KUKA KRL program: Milling_2_222.src

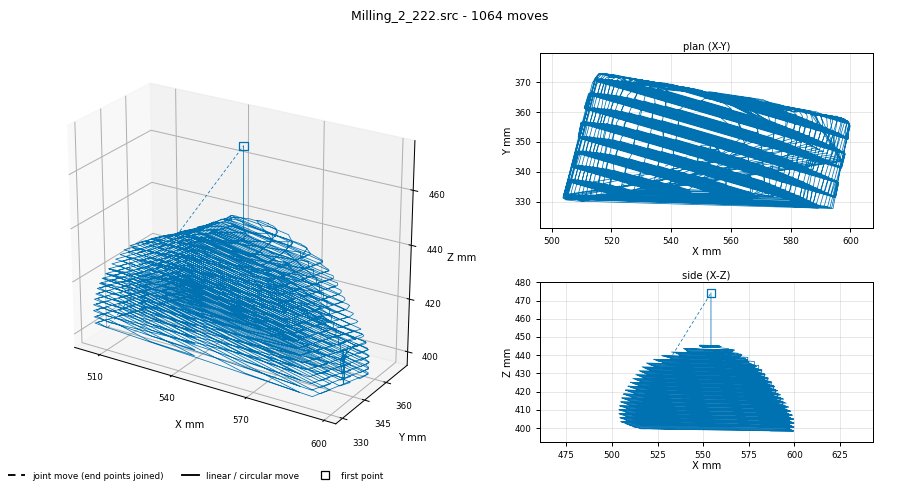
[picture p0: tool path of Milling_2_222.src, 1064 of 1066 moves have a stored position in this frame; points joined in program order, loops and branches not executed]
&ACCESS RVP
&REL 1
&PARAM TEMPLATE = C:\KRC\Roboter\Template\vorgabe
&PARAM EDITMASK = *
DEF Milling_2_222 ( )


;FOLD INI
;FOLD BASISTECH INI
GLOBAL INTERRUPT DECL 3 WHEN $STOPMESS==TRUE DO IR_STOPM ( )
INTERRUPT ON 3
BAS (#INITMOV,0 )
;ENDFOLD (BASISTECH INI)
;ENDFOLD (INI)

;FOLD STARTPOSITION - BASE IS 0, TOOL IS 5, SPEED IS 15%, POSITION IS A1 5,A2 -90,A3 100,A4 5,A5 -10,A6 -5,E1 0,E2 0,E3 0,E4 0
$BWDSTART = FALSE
PDAT_ACT = {VEL 15,ACC 100,APO_DIST 50}
FDAT_ACT = {TOOL_NO 5,BASE_NO 0,IPO_FRAME #BASE}
BAS (#PTP_PARAMS,15)
PTP  {A1 5,A2 -90,A3 100,A4 5,A5 -10,A6 -5,E1 0,E2 0,E3 0,E4 0}
;ENDFOLD

;FOLD LIN SPEED IS 0.1 m/sec, INTERPOLATION SETTINGS IN FOLD
$VEL.CP=0.1
$ADVANCE=3
;ENDFOLD

;FOLD COMMANDS IN FOLD. SELECT EDIT/FOLDS/OPEN ALL FOLDS TO DISPLAY
BAS(#VEL_PTP,2)
PTP {X 554.276, Y 348.908, Z 474.151, A -110.612, B 84.801, C -94.37, E1 0, E2 0, E3 0, E4 0, S 'B010'}
$VEL.CP=0.012
LIN {X 554.276, Y 348.908, Z 444.151, A -110.612, B 84.801, C -94.37, E1 0, E2 0, E3 0, E4 0}
LIN {X 558.607, Y 344.235, Z 444.41, A -110.612, B 84.801, C -94.37, E1 0, E2 0, E3 0, E4 0}
LIN {X 558.405, Y 342.44, Z 444.57, A -110.612, B 84.801, C -94.37, E1 0, E2 0, E3 0, E4 0}
LIN {X 559.721, Y 340.767, Z 444.67, A -110.612, B 84.801, C -94.37, E1 0, E2 0, E3 0, E4 0}
LIN {X 559.873, Y 339.853, Z 444.743, A -110.612, B 84.801, C -94.37, E1 0, E2 0, E3 0, E4 0}
LIN {X 557.875, Y 337.185, Z 445.034, A -110.612, B 84.801, C -94.37, E1 0, E2 0, E3 0, E4 0}
LIN {X 558.814, Y 334.358, Z 445.245, A -110.612, B 84.801, C -94.37, E1 0, E2 0, E3 0, E4 0}
LIN {X 549.81, Y 334.655, Z 445.508, A -110.612, B 84.801, C -94.37, E1 0, E2 0, E3 0, E4 0}
LIN {X 548.065, Y 334.808, Z 445.551, A -110.612, B 84.801, C -94.37, E1 0, E2 0, E3 0, E4 0}
LIN {X 547.985, Y 340.162, Z 445.098, A -110.612, B 84.801, C -94.37, E1 0, E2 0, E3 0, E4 0}
LIN {X 547.942, Y 340.376, Z 445.081, A -110.612, B 84.801, C -94.37, E1 0, E2 0, E3 0, E4 0}
LIN {X 549.959, Y 348.904, Z 444.29, A -110.612, B 84.801, C -94.37, E1 0, E2 0, E3 0, E4 0}
LIN {X 554.276, Y 348.908, Z 444.151, A -110.612, B 84.801, C -94.37, E1 0, E2 0, E3 0, E4 0}
LIN {X 556.311, Y 346.712, Z 444.273, A -110.612, B 84.801, C -94.37, E1 0, E2 0, E3 0, E4 0}
LIN {X 549.895, Y 348.583, Z 444.319, A -110.612, B 84.801, C -94.37, E1 0, E2 0, E3 0, E4 0}
LIN {X 548.877, Y 343.693, Z 444.768, A -110.612, B 84.801, C -94.37, E1 0, E2 0, E3 0, E4 0}
LIN {X 559.743, Y 340.524, Z 444.69, A -110.612, B 84.801, C -94.37, E1 0, E2 0, E3 0, E4 0}
LIN {X 558.354, Y 335.742, Z 445.142, A -110.612, B 84.801, C -94.37, E1 0, E2 0, E3 0, E4 0}
LIN {X 547.877, Y 338.798, Z 445.217, A -110.612, B 84.801, C -94.37, E1 0, E2 0, E3 0, E4 0}
LIN {X 563.989, Y 351.833, Z 443.591, A -110.612, B 84.801, C -94.37, E1 0, E2 0, E3 0, E4 0}
LIN {X 563.919, Y 351.649, Z 441.427, A -110.612, B 84.801, C -94.37, E1 0, E2 0, E3 0, E4 0}
LIN {X 565.535, Y 346.359, Z 441.825, A -110.612, B 84.801, C -94.37, E1 0, E2 0, E3 0, E4 0}
LIN {X 565.665, Y 346.192, Z 441.835, A -110.612, B 84.801, C -94.37, E1 0, E2 0, E3 0, E4 0}
LIN {X 567.236, Y 333.139, Z 442.897, A -110.612, B 84.801, C -94.37, E1 0, E2 0, E3 0, E4 0}
LIN {X 541.312, Y 334.209, Z 443.636, A -110.612, B 84.801, C -94.37, E1 0, E2 0, E3 0, E4 0}
LIN {X 539.137, Y 334.152, Z 443.71, A -110.612, B 84.801, C -94.37, E1 0, E2 0, E3 0, E4 0}
LIN {X 541.372, Y 343.839, Z 442.814, A -110.612, B 84.801, C -94.37, E1 0, E2 0, E3 0, E4 0}
LIN {X 540.702, Y 345.693, Z 442.677, A -110.612, B 84.801, C -94.37, E1 0, E2 0, E3 0, E4 0}
LIN {X 540.663, Y 347.231, Z 442.548, A -110.612, B 84.801, C -94.37, E1 0, E2 0, E3 0, E4 0}
LIN {X 540.807, Y 347.464, Z 442.523, A -110.612, B 84.801, C -94.37, E1 0, E2 0, E3 0, E4 0}
LIN {X 540.755, Y 349.434, Z 442.357, A -110.612, B 84.801, C -94.37, E1 0, E2 0, E3 0, E4 0}
LIN {X 541.559, Y 350.645, Z 442.228, A -110.612, B 84.801, C -94.37, E1 0, E2 0, E3 0, E4 0}
LIN {X 542.49, Y 357.115, Z 441.648, A -110.612, B 84.801, C -94.37, E1 0, E2 0, E3 0, E4 0}
LIN {X 543.459, Y 357.876, Z 441.552, A -110.612, B 84.801, C -94.37, E1 0, E2 0, E3 0, E4 0}
LIN {X 543.538, Y 358.445, Z 441.501, A -110.612, B 84.801, C -94.37, E1 0, E2 0, E3 0, E4 0}
LIN {X 541.559, Y 360.385, Z 441.399, A -110.612, B 84.801, C -94.37, E1 0, E2 0, E3 0, E4 0}
LIN {X 543.39, Y 361.216, Z 441.27, A -110.612, B 84.801, C -94.37, E1 0, E2 0, E3 0, E4 0}
LIN {X 544.179, Y 362.266, Z 441.155, A -110.612, B 84.801, C -94.37, E1 0, E2 0, E3 0, E4 0}
LIN {X 544.202, Y 362.541, Z 441.131, A -110.612, B 84.801, C -94.37, E1 0, E2 0, E3 0, E4 0}
LIN {X 544.848, Y 362.434, Z 441.119, A -110.612, B 84.801, C -94.37, E1 0, E2 0, E3 0, E4 0}
LIN {X 547.986, Y 363.741, Z 440.907, A -110.612, B 84.801, C -94.37, E1 0, E2 0, E3 0, E4 0}
LIN {X 548.585, Y 363.499, Z 440.909, A -110.612, B 84.801, C -94.37, E1 0, E2 0, E3 0, E4 0}
LIN {X 549.994, Y 363.669, Z 440.849, A -110.612, B 84.801, C -94.37, E1 0, E2 0, E3 0, E4 0}
LIN {X 551.281, Y 364.62, Z 440.727, A -110.612, B 84.801, C -94.37, E1 0, E2 0, E3 0, E4 0}
LIN {X 554.079, Y 364.139, Z 440.678, A -110.612, B 84.801, C -94.37, E1 0, E2 0, E3 0, E4 0}
LIN {X 554.813, Y 364.232, Z 440.647, A -110.612, B 84.801, C -94.37, E1 0, E2 0, E3 0, E4 0}
LIN {X 554.86, Y 363.85, Z 440.678, A -110.612, B 84.801, C -94.37, E1 0, E2 0, E3 0, E4 0}
LIN {X 557.614, Y 363.059, Z 440.657, A -110.612, B 84.801, C -94.37, E1 0, E2 0, E3 0, E4 0}
LIN {X 559.744, Y 361.401, Z 440.73, A -110.612, B 84.801, C -94.37, E1 0, E2 0, E3 0, E4 0}
LIN {X 560.566, Y 360.153, Z 440.81, A -110.612, B 84.801, C -94.37, E1 0, E2 0, E3 0, E4 0}
LIN {X 561.613, Y 359.2, Z 440.857, A -110.612, B 84.801, C -94.37, E1 0, E2 0, E3 0, E4 0}
LIN {X 563.919, Y 351.649, Z 441.427, A -110.612, B 84.801, C -94.37, E1 0, E2 0, E3 0, E4 0}
LIN {X 550.229, Y 363.842, Z 440.827, A -110.612, B 84.801, C -94.37, E1 0, E2 0, E3 0, E4 0}
LIN {X 560.058, Y 360.976, Z 440.756, A -110.612, B 84.801, C -94.37, E1 0, E2 0, E3 0, E4 0}
LIN {X 563.393, Y 354.816, Z 441.174, A -110.612, B 84.801, C -94.37, E1 0, E2 0, E3 0, E4 0}
LIN {X 542.631, Y 360.871, Z 441.323, A -110.612, B 84.801, C -94.37, E1 0, E2 0, E3 0, E4 0}
LIN {X 542.344, Y 355.768, Z 441.767, A -110.612, B 84.801, C -94.37, E1 0, E2 0, E3 0, E4 0}
LIN {X 565.078, Y 349.137, Z 441.603, A -110.612, B 84.801, C -94.37, E1 0, E2 0, E3 0, E4 0}
LIN {X 565.885, Y 343.715, Z 442.039, A -110.612, B 84.801, C -94.37, E1 0, E2 0, E3 0, E4 0}
LIN {X 541.583, Y 350.803, Z 442.214, A -110.612, B 84.801, C -94.37, E1 0, E2 0, E3 0, E4 0}
LIN {X 540.685, Y 345.878, Z 442.662, A -110.612, B 84.801, C -94.37, E1 0, E2 0, E3 0, E4 0}
LIN {X 566.796, Y 338.262, Z 442.474, A -110.612, B 84.801, C -94.37, E1 0, E2 0, E3 0, E4 0}
LIN {X 566.499, Y 333.162, Z 442.918, A -110.612, B 84.801, C -94.37, E1 0, E2 0, E3 0, E4 0}
LIN {X 540.83, Y 340.648, Z 443.103, A -110.612, B 84.801, C -94.37, E1 0, E2 0, E3 0, E4 0}
LIN {X 539.697, Y 335.792, Z 443.553, A -110.612, B 84.801, C -94.37, E1 0, E2 0, E3 0, E4 0}
LIN {X 545.888, Y 333.986, Z 443.508, A -110.612, B 84.801, C -94.37, E1 0, E2 0, E3 0, E4 0}
LIN {X 569.078, Y 353.533, Z 441.101, A -110.612, B 84.801, C -94.37, E1 0, E2 0, E3 0, E4 0}
LIN {X 569.009, Y 353.348, Z 438.936, A -110.612, B 84.801, C -94.37, E1 0, E2 0, E3 0, E4 0}
LIN {X 570.01, Y 350.644, Z 439.134, A -110.612, B 84.801, C -94.37, E1 0, E2 0, E3 0, E4 0}
LIN {X 571.217, Y 336.984, Z 440.258, A -110.612, B 84.801, C -94.37, E1 0, E2 0, E3 0, E4 0}
LIN {X 570.966, Y 336.181, Z 440.335, A -110.612, B 84.801, C -94.37, E1 0, E2 0, E3 0, E4 0}
LIN {X 570.983, Y 334.774, Z 440.454, A -110.612, B 84.801, C -94.37, E1 0, E2 0, E3 0, E4 0}
LIN {X 570.338, Y 332.582, Z 440.661, A -110.612, B 84.801, C -94.37, E1 0, E2 0, E3 0, E4 0}
LIN {X 534.018, Y 333.771, Z 441.723, A -110.612, B 84.801, C -94.37, E1 0, E2 0, E3 0, E4 0}
LIN {X 532.644, Y 333.742, Z 441.77, A -110.612, B 84.801, C -94.37, E1 0, E2 0, E3 0, E4 0}
LIN {X 535.31, Y 339.493, Z 441.195, A -110.612, B 84.801, C -94.37, E1 0, E2 0, E3 0, E4 0}
LIN {X 535.287, Y 341.092, Z 441.059, A -110.612, B 84.801, C -94.37, E1 0, E2 0, E3 0, E4 0}
LIN {X 537.309, Y 348.411, Z 440.371, A -110.612, B 84.801, C -94.37, E1 0, E2 0, E3 0, E4 0}
LIN {X 537.606, Y 348.945, Z 440.316, A -110.612, B 84.801, C -94.37, E1 0, E2 0, E3 0, E4 0}
LIN {X 537.307, Y 354.669, Z 439.838, A -110.612, B 84.801, C -94.37, E1 0, E2 0, E3 0, E4 0}
LIN {X 536.893, Y 356.232, Z 439.719, A -110.612, B 84.801, C -94.37, E1 0, E2 0, E3 0, E4 0}
LIN {X 536.949, Y 357.185, Z 439.636, A -110.612, B 84.801, C -94.37, E1 0, E2 0, E3 0, E4 0}
LIN {X 537.165, Y 357.599, Z 439.593, A -110.612, B 84.801, C -94.37, E1 0, E2 0, E3 0, E4 0}
LIN {X 538.343, Y 363.903, Z 439.019, A -110.612, B 84.801, C -94.37, E1 0, E2 0, E3 0, E4 0}
LIN {X 538.336, Y 363.912, Z 439.018, A -110.612, B 84.801, C -94.37, E1 0, E2 0, E3 0, E4 0}
LIN {X 537.831, Y 366.807, Z 438.788, A -110.612, B 84.801, C -94.37, E1 0, E2 0, E3 0, E4 0}
LIN {X 537.936, Y 366.972, Z 438.77, A -110.612, B 84.801, C -94.37, E1 0, E2 0, E3 0, E4 0}
LIN {X 539.378, Y 367.681, Z 438.664, A -110.612, B 84.801, C -94.37, E1 0, E2 0, E3 0, E4 0}
LIN {X 552.236, Y 366.051, Z 438.391, A -110.612, B 84.801, C -94.37, E1 0, E2 0, E3 0, E4 0}
LIN {X 554.008, Y 366.638, Z 438.284, A -110.612, B 84.801, C -94.37, E1 0, E2 0, E3 0, E4 0}
LIN {X 562.727, Y 364.468, Z 438.19, A -110.612, B 84.801, C -94.37, E1 0, E2 0, E3 0, E4 0}
LIN {X 566.199, Y 360.577, Z 438.41, A -110.612, B 84.801, C -94.37, E1 0, E2 0, E3 0, E4 0}
LIN {X 567.699, Y 358.885, Z 438.506, A -110.612, B 84.801, C -94.37, E1 0, E2 0, E3 0, E4 0}
LIN {X 569.005, Y 355.632, Z 438.741, A -110.612, B 84.801, C -94.37, E1 0, E2 0, E3 0, E4 0}
LIN {X 569.009, Y 353.348, Z 438.936, A -110.612, B 84.801, C -94.37, E1 0, E2 0, E3 0, E4 0}
LIN {X 567.859, Y 358.496, Z 438.534, A -110.612, B 84.801, C -94.37, E1 0, E2 0, E3 0, E4 0}
LIN {X 538.218, Y 367.141, Z 438.747, A -110.612, B 84.801, C -94.37, E1 0, E2 0, E3 0, E4 0}
LIN {X 538.244, Y 361.946, Z 439.189, A -110.612, B 84.801, C -94.37, E1 0, E2 0, E3 0, E4 0}
LIN {X 569.164, Y 352.928, Z 438.966, A -110.612, B 84.801, C -94.37, E1 0, E2 0, E3 0, E4 0}
LIN {X 570.368, Y 347.39, Z 439.4, A -110.612, B 84.801, C -94.37, E1 0, E2 0, E3 0, E4 0}
LIN {X 536.951, Y 357.136, Z 439.64, A -110.612, B 84.801, C -94.37, E1 0, E2 0, E3 0, E4 0}
LIN {X 537.304, Y 351.846, Z 440.079, A -110.612, B 84.801, C -94.37, E1 0, E2 0, E3 0, E4 0}
LIN {X 570.875, Y 342.055, Z 439.838, A -110.612, B 84.801, C -94.37, E1 0, E2 0, E3 0, E4 0}
LIN {X 571.155, Y 336.786, Z 440.277, A -110.612, B 84.801, C -94.37, E1 0, E2 0, E3 0, E4 0}
LIN {X 536.952, Y 346.762, Z 440.523, A -110.612, B 84.801, C -94.37, E1 0, E2 0, E3 0, E4 0}
LIN {X 535.523, Y 341.992, Z 440.975, A -110.612, B 84.801, C -94.37, E1 0, E2 0, E3 0, E4 0}
LIN {X 566.961, Y 332.823, Z 440.749, A -110.612, B 84.801, C -94.37, E1 0, E2 0, E3 0, E4 0}
LIN {X 546.398, Y 333.633, Z 441.339, A -110.612, B 84.801, C -94.37, E1 0, E2 0, E3 0, E4 0}
LIN {X 534.432, Y 337.123, Z 441.425, A -110.612, B 84.801, C -94.37, E1 0, E2 0, E3 0, E4 0}
LIN {X 574.468, Y 352.804, Z 438.807, A -110.612, B 84.801, C -94.37, E1 0, E2 0, E3 0, E4 0}
LIN {X 574.398, Y 352.62, Z 436.642, A -110.612, B 84.801, C -94.37, E1 0, E2 0, E3 0, E4 0}
LIN {X 574.985, Y 358.624, Z 436.112, A -110.612, B 84.801, C -94.37, E1 0, E2 0, E3 0, E4 0}
LIN {X 569.893, Y 363.529, Z 435.858, A -110.612, B 84.801, C -94.37, E1 0, E2 0, E3 0, E4 0}
LIN {X 568.224, Y 364.067, Z 435.865, A -110.612, B 84.801, C -94.37, E1 0, E2 0, E3 0, E4 0}
LIN {X 568.037, Y 364.329, Z 435.849, A -110.612, B 84.801, C -94.37, E1 0, E2 0, E3 0, E4 0}
LIN {X 567.581, Y 364.537, Z 435.846, A -110.612, B 84.801, C -94.37, E1 0, E2 0, E3 0, E4 0}
LIN {X 554.164, Y 366.346, Z 436.121, A -110.612, B 84.801, C -94.37, E1 0, E2 0, E3 0, E4 0}
LIN {X 553.733, Y 366.168, Z 436.15, A -110.612, B 84.801, C -94.37, E1 0, E2 0, E3 0, E4 0}
LIN {X 542.465, Y 368.047, Z 436.351, A -110.612, B 84.801, C -94.37, E1 0, E2 0, E3 0, E4 0}
LIN {X 540.849, Y 369.238, Z 436.301, A -110.612, B 84.801, C -94.37, E1 0, E2 0, E3 0, E4 0}
LIN {X 538.504, Y 369.469, Z 436.357, A -110.612, B 84.801, C -94.37, E1 0, E2 0, E3 0, E4 0}
LIN {X 537.187, Y 369.143, Z 436.427, A -110.612, B 84.801, C -94.37, E1 0, E2 0, E3 0, E4 0}
LIN {X 535.889, Y 368.249, Z 436.545, A -110.612, B 84.801, C -94.37, E1 0, E2 0, E3 0, E4 0}
LIN {X 534.308, Y 366.474, Z 436.746, A -110.612, B 84.801, C -94.37, E1 0, E2 0, E3 0, E4 0}
LIN {X 534.281, Y 366.405, Z 436.753, A -110.612, B 84.801, C -94.37, E1 0, E2 0, E3 0, E4 0}
LIN {X 534.584, Y 363.066, Z 437.028, A -110.612, B 84.801, C -94.37, E1 0, E2 0, E3 0, E4 0}
LIN {X 534.095, Y 360.828, Z 437.234, A -110.612, B 84.801, C -94.37, E1 0, E2 0, E3 0, E4 0}
LIN {X 533.835, Y 360.635, Z 437.259, A -110.612, B 84.801, C -94.37, E1 0, E2 0, E3 0, E4 0}
LIN {X 533.475, Y 357.247, Z 437.559, A -110.612, B 84.801, C -94.37, E1 0, E2 0, E3 0, E4 0}
LIN {X 533.725, Y 356.099, Z 437.649, A -110.612, B 84.801, C -94.37, E1 0, E2 0, E3 0, E4 0}
LIN {X 530.786, Y 342.023, Z 438.942, A -110.612, B 84.801, C -94.37, E1 0, E2 0, E3 0, E4 0}
LIN {X 528.148, Y 336.133, Z 439.528, A -110.612, B 84.801, C -94.37, E1 0, E2 0, E3 0, E4 0}
LIN {X 527.371, Y 333.264, Z 439.797, A -110.612, B 84.801, C -94.37, E1 0, E2 0, E3 0, E4 0}
LIN {X 572.535, Y 332.154, Z 438.445, A -110.612, B 84.801, C -94.37, E1 0, E2 0, E3 0, E4 0}
LIN {X 574.204, Y 350.632, Z 436.818, A -110.612, B 84.801, C -94.37, E1 0, E2 0, E3 0, E4 0}
LIN {X 574.398, Y 352.62, Z 436.642, A -110.612, B 84.801, C -94.37, E1 0, E2 0, E3 0, E4 0}
LIN {X 571.376, Y 362.452, Z 435.902, A -110.612, B 84.801, C -94.37, E1 0, E2 0, E3 0, E4 0}
LIN {X 561.721, Y 365.268, Z 435.971, A -110.612, B 84.801, C -94.37, E1 0, E2 0, E3 0, E4 0}
LIN {X 561.675, Y 365.282, Z 435.971, A -110.612, B 84.801, C -94.37, E1 0, E2 0, E3 0, E4 0}
LIN {X 535.453, Y 367.743, Z 436.602, A -110.612, B 84.801, C -94.37, E1 0, E2 0, E3 0, E4 0}
LIN {X 574.931, Y 356.229, Z 436.318, A -110.612, B 84.801, C -94.37, E1 0, E2 0, E3 0, E4 0}
LIN {X 574.139, Y 351.273, Z 436.765, A -110.612, B 84.801, C -94.37, E1 0, E2 0, E3 0, E4 0}
LIN {X 534.55, Y 362.819, Z 437.05, A -110.612, B 84.801, C -94.37, E1 0, E2 0, E3 0, E4 0}
LIN {X 533.571, Y 357.917, Z 437.499, A -110.612, B 84.801, C -94.37, E1 0, E2 0, E3 0, E4 0}
LIN {X 574.308, Y 346.036, Z 437.206, A -110.612, B 84.801, C -94.37, E1 0, E2 0, E3 0, E4 0}
LIN {X 573.943, Y 340.956, Z 437.65, A -110.612, B 84.801, C -94.37, E1 0, E2 0, E3 0, E4 0}
LIN {X 533.122, Y 352.862, Z 437.944, A -110.612, B 84.801, C -94.37, E1 0, E2 0, E3 0, E4 0}
LIN {X 532.259, Y 347.926, Z 438.392, A -110.612, B 84.801, C -94.37, E1 0, E2 0, E3 0, E4 0}
LIN {X 573.267, Y 335.966, Z 438.097, A -110.612, B 84.801, C -94.37, E1 0, E2 0, E3 0, E4 0}
LIN {X 567.221, Y 332.542, Z 438.582, A -110.612, B 84.801, C -94.37, E1 0, E2 0, E3 0, E4 0}
LIN {X 530.884, Y 343.14, Z 438.843, A -110.612, B 84.801, C -94.37, E1 0, E2 0, E3 0, E4 0}
LIN {X 529.176, Y 338.451, Z 439.297, A -110.612, B 84.801, C -94.37, E1 0, E2 0, E3 0, E4 0}
LIN {X 546.678, Y 333.347, Z 439.171, A -110.612, B 84.801, C -94.37, E1 0, E2 0, E3 0, E4 0}
LIN {X 528.874, Y 333.353, Z 439.741, A -110.612, B 84.801, C -94.37, E1 0, E2 0, E3 0, E4 0}
LIN {X 527.487, Y 333.757, Z 439.751, A -110.612, B 84.801, C -94.37, E1 0, E2 0, E3 0, E4 0}
LIN {X 578.084, Y 351.918, Z 436.584, A -110.612, B 84.801, C -94.37, E1 0, E2 0, E3 0, E4 0}
LIN {X 578.015, Y 351.733, Z 434.419, A -110.612, B 84.801, C -94.37, E1 0, E2 0, E3 0, E4 0}
LIN {X 574.255, Y 331.838, Z 436.234, A -110.612, B 84.801, C -94.37, E1 0, E2 0, E3 0, E4 0}
LIN {X 523.53, Y 333.036, Z 437.756, A -110.612, B 84.801, C -94.37, E1 0, E2 0, E3 0, E4 0}
LIN {X 522.764, Y 332.973, Z 437.786, A -110.612, B 84.801, C -94.37, E1 0, E2 0, E3 0, E4 0}
LIN {X 525.236, Y 343.034, Z 436.85, A -110.612, B 84.801, C -94.37, E1 0, E2 0, E3 0, E4 0}
LIN {X 526.652, Y 345.685, Z 436.579, A -110.612, B 84.801, C -94.37, E1 0, E2 0, E3 0, E4 0}
LIN {X 531.3, Y 365.618, Z 434.733, A -110.612, B 84.801, C -94.37, E1 0, E2 0, E3 0, E4 0}
LIN {X 532.889, Y 368.619, Z 434.426, A -110.612, B 84.801, C -94.37, E1 0, E2 0, E3 0, E4 0}
LIN {X 535.381, Y 369.826, Z 434.244, A -110.612, B 84.801, C -94.37, E1 0, E2 0, E3 0, E4 0}
LIN {X 537.674, Y 369.756, Z 434.176, A -110.612, B 84.801, C -94.37, E1 0, E2 0, E3 0, E4 0}
LIN {X 541.064, Y 368.842, Z 434.145, A -110.612, B 84.801, C -94.37, E1 0, E2 0, E3 0, E4 0}
LIN {X 542.193, Y 367.93, Z 434.187, A -110.612, B 84.801, C -94.37, E1 0, E2 0, E3 0, E4 0}
LIN {X 551.391, Y 366.541, Z 434.011, A -110.612, B 84.801, C -94.37, E1 0, E2 0, E3 0, E4 0}
LIN {X 552.803, Y 366.842, Z 433.94, A -110.612, B 84.801, C -94.37, E1 0, E2 0, E3 0, E4 0}
LIN {X 570.771, Y 364.151, Z 433.593, A -110.612, B 84.801, C -94.37, E1 0, E2 0, E3 0, E4 0}
LIN {X 578.179, Y 360.934, Z 433.63, A -110.612, B 84.801, C -94.37, E1 0, E2 0, E3 0, E4 0}
LIN {X 578.619, Y 360.438, Z 433.658, A -110.612, B 84.801, C -94.37, E1 0, E2 0, E3 0, E4 0}
LIN {X 579.316, Y 359.01, Z 433.758, A -110.612, B 84.801, C -94.37, E1 0, E2 0, E3 0, E4 0}
LIN {X 579.339, Y 358.741, Z 433.78, A -110.612, B 84.801, C -94.37, E1 0, E2 0, E3 0, E4 0}
LIN {X 578.015, Y 351.733, Z 434.419, A -110.612, B 84.801, C -94.37, E1 0, E2 0, E3 0, E4 0}
LIN {X 578.767, Y 360.092, Z 433.683, A -110.612, B 84.801, C -94.37, E1 0, E2 0, E3 0, E4 0}
LIN {X 561.03, Y 365.265, Z 433.811, A -110.612, B 84.801, C -94.37, E1 0, E2 0, E3 0, E4 0}
LIN {X 532.693, Y 368.343, Z 434.456, A -110.612, B 84.801, C -94.37, E1 0, E2 0, E3 0, E4 0}
LIN {X 578.339, Y 355.03, Z 434.128, A -110.612, B 84.801, C -94.37, E1 0, E2 0, E3 0, E4 0}
LIN {X 577.543, Y 350.075, Z 434.575, A -110.612, B 84.801, C -94.37, E1 0, E2 0, E3 0, E4 0}
LIN {X 530.911, Y 363.676, Z 434.911, A -110.612, B 84.801, C -94.37, E1 0, E2 0, E3 0, E4 0}
LIN {X 529.165, Y 358.998, Z 435.365, A -110.612, B 84.801, C -94.37, E1 0, E2 0, E3 0, E4 0}
LIN {X 576.615, Y 345.159, Z 435.023, A -110.612, B 84.801, C -94.37, E1 0, E2 0, E3 0, E4 0}
LIN {X 575.918, Y 340.175, Z 435.47, A -110.612, B 84.801, C -94.37, E1 0, E2 0, E3 0, E4 0}
LIN {X 528.335, Y 354.053, Z 435.813, A -110.612, B 84.801, C -94.37, E1 0, E2 0, E3 0, E4 0}
LIN {X 527.42, Y 349.133, Z 436.261, A -110.612, B 84.801, C -94.37, E1 0, E2 0, E3 0, E4 0}
LIN {X 574.963, Y 335.266, Z 435.919, A -110.612, B 84.801, C -94.37, E1 0, E2 0, E3 0, E4 0}
LIN {X 567.23, Y 332.335, Z 436.416, A -110.612, B 84.801, C -94.37, E1 0, E2 0, E3 0, E4 0}
LIN {X 525.837, Y 344.408, Z 436.714, A -110.612, B 84.801, C -94.37, E1 0, E2 0, E3 0, E4 0}
LIN {X 524.56, Y 339.593, Z 437.165, A -110.612, B 84.801, C -94.37, E1 0, E2 0, E3 0, E4 0}
LIN {X 546.693, Y 333.138, Z 437.006, A -110.612, B 84.801, C -94.37, E1 0, E2 0, E3 0, E4 0}
LIN {X 528.865, Y 333.151, Z 437.576, A -110.612, B 84.801, C -94.37, E1 0, E2 0, E3 0, E4 0}
LIN {X 523.143, Y 334.819, Z 437.617, A -110.612, B 84.801, C -94.37, E1 0, E2 0, E3 0, E4 0}
LIN {X 580.468, Y 351.172, Z 434.388, A -110.612, B 84.801, C -94.37, E1 0, E2 0, E3 0, E4 0}
LIN {X 580.398, Y 350.988, Z 432.223, A -110.612, B 84.801, C -94.37, E1 0, E2 0, E3 0, E4 0}
LIN {X 575.978, Y 331.564, Z 434.019, A -110.612, B 84.801, C -94.37, E1 0, E2 0, E3 0, E4 0}
LIN {X 521.035, Y 332.721, Z 435.68, A -110.612, B 84.801, C -94.37, E1 0, E2 0, E3 0, E4 0}
LIN {X 518.901, Y 332.776, Z 435.744, A -110.612, B 84.801, C -94.37, E1 0, E2 0, E3 0, E4 0}
LIN {X 520.72, Y 340.63, Z 435.017, A -110.612, B 84.801, C -94.37, E1 0, E2 0, E3 0, E4 0}
LIN {X 520.834, Y 340.798, Z 434.999, A -110.612, B 84.801, C -94.37, E1 0, E2 0, E3 0, E4 0}
LIN {X 520.518, Y 343.145, Z 434.809, A -110.612, B 84.801, C -94.37, E1 0, E2 0, E3 0, E4 0}
LIN {X 523.407, Y 351.6, Z 433.996, A -110.612, B 84.801, C -94.37, E1 0, E2 0, E3 0, E4 0}
LIN {X 524.017, Y 352.182, Z 433.927, A -110.612, B 84.801, C -94.37, E1 0, E2 0, E3 0, E4 0}
LIN {X 524.237, Y 355.868, Z 433.606, A -110.612, B 84.801, C -94.37, E1 0, E2 0, E3 0, E4 0}
LIN {X 529.406, Y 368.041, Z 432.404, A -110.612, B 84.801, C -94.37, E1 0, E2 0, E3 0, E4 0}
LIN {X 531.28, Y 369.724, Z 432.201, A -110.612, B 84.801, C -94.37, E1 0, E2 0, E3 0, E4 0}
LIN {X 532.966, Y 370.274, Z 432.1, A -110.612, B 84.801, C -94.37, E1 0, E2 0, E3 0, E4 0}
LIN {X 540.143, Y 369.059, Z 431.974, A -110.612, B 84.801, C -94.37, E1 0, E2 0, E3 0, E4 0}
LIN {X 540.354, Y 368.938, Z 431.977, A -110.612, B 84.801, C -94.37, E1 0, E2 0, E3 0, E4 0}
LIN {X 541.511, Y 368.887, Z 431.944, A -110.612, B 84.801, C -94.37, E1 0, E2 0, E3 0, E4 0}
LIN {X 542.437, Y 368.241, Z 431.97, A -110.612, B 84.801, C -94.37, E1 0, E2 0, E3 0, E4 0}
LIN {X 543.867, Y 368.523, Z 431.9, A -110.612, B 84.801, C -94.37, E1 0, E2 0, E3 0, E4 0}
LIN {X 547.54, Y 366.999, Z 431.912, A -110.612, B 84.801, C -94.37, E1 0, E2 0, E3 0, E4 0}
LIN {X 551.439, Y 366.924, Z 431.794, A -110.612, B 84.801, C -94.37, E1 0, E2 0, E3 0, E4 0}
LIN {X 551.993, Y 366.678, Z 431.797, A -110.612, B 84.801, C -94.37, E1 0, E2 0, E3 0, E4 0}
LIN {X 569.024, Y 364.084, Z 431.472, A -110.612, B 84.801, C -94.37, E1 0, E2 0, E3 0, E4 0}
LIN {X 569.195, Y 364.114, Z 431.464, A -110.612, B 84.801, C -94.37, E1 0, E2 0, E3 0, E4 0}
LIN {X 576.4, Y 362.509, Z 431.37, A -110.612, B 84.801, C -94.37, E1 0, E2 0, E3 0, E4 0}
LIN {X 576.626, Y 362.397, Z 431.372, A -110.612, B 84.801, C -94.37, E1 0, E2 0, E3 0, E4 0}
LIN {X 576.764, Y 362.414, Z 431.367, A -110.612, B 84.801, C -94.37, E1 0, E2 0, E3 0, E4 0}
LIN {X 580.278, Y 360.239, Z 431.439, A -110.612, B 84.801, C -94.37, E1 0, E2 0, E3 0, E4 0}
LIN {X 580.976, Y 360.034, Z 431.434, A -110.612, B 84.801, C -94.37, E1 0, E2 0, E3 0, E4 0}
LIN {X 582.145, Y 358.757, Z 431.506, A -110.612, B 84.801, C -94.37, E1 0, E2 0, E3 0, E4 0}
LIN {X 582.151, Y 358.689, Z 431.511, A -110.612, B 84.801, C -94.37, E1 0, E2 0, E3 0, E4 0}
LIN {X 580.398, Y 350.988, Z 432.223, A -110.612, B 84.801, C -94.37, E1 0, E2 0, E3 0, E4 0}
LIN {X 560.468, Y 365.225, Z 431.649, A -110.612, B 84.801, C -94.37, E1 0, E2 0, E3 0, E4 0}
LIN {X 581.97, Y 358.954, Z 431.495, A -110.612, B 84.801, C -94.37, E1 0, E2 0, E3 0, E4 0}
LIN {X 580.949, Y 354.064, Z 431.944, A -110.612, B 84.801, C -94.37, E1 0, E2 0, E3 0, E4 0}
LIN {X 530.225, Y 368.858, Z 432.308, A -110.612, B 84.801, C -94.37, E1 0, E2 0, E3 0, E4 0}
LIN {X 527.54, Y 364.454, Z 432.769, A -110.612, B 84.801, C -94.37, E1 0, E2 0, E3 0, E4 0}
LIN {X 579.85, Y 349.198, Z 432.393, A -110.612, B 84.801, C -94.37, E1 0, E2 0, E3 0, E4 0}
LIN {X 578.612, Y 344.372, Z 432.844, A -110.612, B 84.801, C -94.37, E1 0, E2 0, E3 0, E4 0}
LIN {X 525.917, Y 359.741, Z 433.223, A -110.612, B 84.801, C -94.37, E1 0, E2 0, E3 0, E4 0}
LIN {X 524.197, Y 355.055, Z 433.677, A -110.612, B 84.801, C -94.37, E1 0, E2 0, E3 0, E4 0}
LIN {X 577.658, Y 339.463, Z 433.292, A -110.612, B 84.801, C -94.37, E1 0, E2 0, E3 0, E4 0}
LIN {X 576.646, Y 334.571, Z 433.741, A -110.612, B 84.801, C -94.37, E1 0, E2 0, E3 0, E4 0}
LIN {X 522.84, Y 350.264, Z 434.128, A -110.612, B 84.801, C -94.37, E1 0, E2 0, E3 0, E4 0}
LIN {X 521.544, Y 345.455, Z 434.58, A -110.612, B 84.801, C -94.37, E1 0, E2 0, E3 0, E4 0}
LIN {X 567.264, Y 332.12, Z 434.251, A -110.612, B 84.801, C -94.37, E1 0, E2 0, E3 0, E4 0}
LIN {X 546.731, Y 332.922, Z 434.84, A -110.612, B 84.801, C -94.37, E1 0, E2 0, E3 0, E4 0}
LIN {X 520.683, Y 340.519, Z 435.027, A -110.612, B 84.801, C -94.37, E1 0, E2 0, E3 0, E4 0}
LIN {X 519.275, Y 335.743, Z 435.479, A -110.612, B 84.801, C -94.37, E1 0, E2 0, E3 0, E4 0}
LIN {X 528.883, Y 332.941, Z 435.41, A -110.612, B 84.801, C -94.37, E1 0, E2 0, E3 0, E4 0}
LIN {X 582.137, Y 350.577, Z 432.202, A -110.612, B 84.801, C -94.37, E1 0, E2 0, E3 0, E4 0}
LIN {X 582.068, Y 350.393, Z 430.037, A -110.612, B 84.801, C -94.37, E1 0, E2 0, E3 0, E4 0}
LIN {X 577.57, Y 331.244, Z 431.812, A -110.612, B 84.801, C -94.37, E1 0, E2 0, E3 0, E4 0}
LIN {X 519.27, Y 332.577, Z 433.566, A -110.612, B 84.801, C -94.37, E1 0, E2 0, E3 0, E4 0}
LIN {X 516.471, Y 332.54, Z 433.659, A -110.612, B 84.801, C -94.37, E1 0, E2 0, E3 0, E4 0}
LIN {X 521.738, Y 356.526, Z 431.447, A -110.612, B 84.801, C -94.37, E1 0, E2 0, E3 0, E4 0}
LIN {X 522.162, Y 357.104, Z 431.385, A -110.612, B 84.801, C -94.37, E1 0, E2 0, E3 0, E4 0}
LIN {X 522.633, Y 358.903, Z 431.216, A -110.612, B 84.801, C -94.37, E1 0, E2 0, E3 0, E4 0}
LIN {X 525.463, Y 365.719, Z 430.545, A -110.612, B 84.801, C -94.37, E1 0, E2 0, E3 0, E4 0}
LIN {X 526.647, Y 366.83, Z 430.413, A -110.612, B 84.801, C -94.37, E1 0, E2 0, E3 0, E4 0}
LIN {X 528.06, Y 369.94, Z 430.103, A -110.612, B 84.801, C -94.37, E1 0, E2 0, E3 0, E4 0}
LIN {X 529.259, Y 370.693, Z 430, A -110.612, B 84.801, C -94.37, E1 0, E2 0, E3 0, E4 0}
LIN {X 532.053, Y 370.536, Z 429.924, A -110.612, B 84.801, C -94.37, E1 0, E2 0, E3 0, E4 0}
LIN {X 532.936, Y 369.925, Z 429.948, A -110.612, B 84.801, C -94.37, E1 0, E2 0, E3 0, E4 0}
LIN {X 533.734, Y 369.748, Z 429.937, A -110.612, B 84.801, C -94.37, E1 0, E2 0, E3 0, E4 0}
LIN {X 535.259, Y 369.982, Z 429.868, A -110.612, B 84.801, C -94.37, E1 0, E2 0, E3 0, E4 0}
LIN {X 539.963, Y 369.103, Z 429.793, A -110.612, B 84.801, C -94.37, E1 0, E2 0, E3 0, E4 0}
LIN {X 541.786, Y 368.061, Z 429.823, A -110.612, B 84.801, C -94.37, E1 0, E2 0, E3 0, E4 0}
LIN {X 542.557, Y 367.997, Z 429.804, A -110.612, B 84.801, C -94.37, E1 0, E2 0, E3 0, E4 0}
LIN {X 543.424, Y 368.55, Z 429.729, A -110.612, B 84.801, C -94.37, E1 0, E2 0, E3 0, E4 0}
LIN {X 551.317, Y 366.87, Z 429.619, A -110.612, B 84.801, C -94.37, E1 0, E2 0, E3 0, E4 0}
LIN {X 551.926, Y 366.297, Z 429.648, A -110.612, B 84.801, C -94.37, E1 0, E2 0, E3 0, E4 0}
LIN {X 553.613, Y 365.853, Z 429.632, A -110.612, B 84.801, C -94.37, E1 0, E2 0, E3 0, E4 0}
LIN {X 556.1, Y 364.537, Z 429.665, A -110.612, B 84.801, C -94.37, E1 0, E2 0, E3 0, E4 0}
LIN {X 556.641, Y 364.535, Z 429.647, A -110.612, B 84.801, C -94.37, E1 0, E2 0, E3 0, E4 0}
LIN {X 558.926, Y 365.163, Z 429.521, A -110.612, B 84.801, C -94.37, E1 0, E2 0, E3 0, E4 0}
LIN {X 559.765, Y 365.162, Z 429.494, A -110.612, B 84.801, C -94.37, E1 0, E2 0, E3 0, E4 0}
LIN {X 560.165, Y 364.978, Z 429.497, A -110.612, B 84.801, C -94.37, E1 0, E2 0, E3 0, E4 0}
LIN {X 562.234, Y 365.034, Z 429.426, A -110.612, B 84.801, C -94.37, E1 0, E2 0, E3 0, E4 0}
LIN {X 567.406, Y 363.847, Z 429.361, A -110.612, B 84.801, C -94.37, E1 0, E2 0, E3 0, E4 0}
LIN {X 567.775, Y 363.945, Z 429.341, A -110.612, B 84.801, C -94.37, E1 0, E2 0, E3 0, E4 0}
LIN {X 578.265, Y 361.313, Z 429.229, A -110.612, B 84.801, C -94.37, E1 0, E2 0, E3 0, E4 0}
LIN {X 578.315, Y 361.327, Z 429.227, A -110.612, B 84.801, C -94.37, E1 0, E2 0, E3 0, E4 0}
LIN {X 578.414, Y 361.275, Z 429.228, A -110.612, B 84.801, C -94.37, E1 0, E2 0, E3 0, E4 0}
LIN {X 582.758, Y 360.509, Z 429.154, A -110.612, B 84.801, C -94.37, E1 0, E2 0, E3 0, E4 0}
LIN {X 583.98, Y 358.533, Z 429.283, A -110.612, B 84.801, C -94.37, E1 0, E2 0, E3 0, E4 0}
LIN {X 582.068, Y 350.393, Z 430.037, A -110.612, B 84.801, C -94.37, E1 0, E2 0, E3 0, E4 0}
LIN {X 583.969, Y 358.166, Z 429.315, A -110.612, B 84.801, C -94.37, E1 0, E2 0, E3 0, E4 0}
LIN {X 560.841, Y 364.911, Z 429.481, A -110.612, B 84.801, C -94.37, E1 0, E2 0, E3 0, E4 0}
LIN {X 527.741, Y 369.378, Z 430.161, A -110.612, B 84.801, C -94.37, E1 0, E2 0, E3 0, E4 0}
LIN {X 582.834, Y 353.31, Z 429.765, A -110.612, B 84.801, C -94.37, E1 0, E2 0, E3 0, E4 0}
LIN {X 581.5, Y 348.512, Z 430.216, A -110.612, B 84.801, C -94.37, E1 0, E2 0, E3 0, E4 0}
LIN {X 525.057, Y 364.974, Z 430.622, A -110.612, B 84.801, C -94.37, E1 0, E2 0, E3 0, E4 0}
LIN {X 523.33, Y 360.291, Z 431.076, A -110.612, B 84.801, C -94.37, E1 0, E2 0, E3 0, E4 0}
LIN {X 580.316, Y 343.67, Z 430.666, A -110.612, B 84.801, C -94.37, E1 0, E2 0, E3 0, E4 0}
LIN {X 579.317, Y 338.775, Z 431.115, A -110.612, B 84.801, C -94.37, E1 0, E2 0, E3 0, E4 0}
LIN {X 521.512, Y 355.634, Z 431.531, A -110.612, B 84.801, C -94.37, E1 0, E2 0, E3 0, E4 0}
LIN {X 520.22, Y 350.824, Z 431.982, A -110.612, B 84.801, C -94.37, E1 0, E2 0, E3 0, E4 0}
LIN {X 578.198, Y 333.914, Z 431.565, A -110.612, B 84.801, C -94.37, E1 0, E2 0, E3 0, E4 0}
LIN {X 567.291, Y 331.908, Z 432.085, A -110.612, B 84.801, C -94.37, E1 0, E2 0, E3 0, E4 0}
LIN {X 519.262, Y 345.916, Z 432.43, A -110.612, B 84.801, C -94.37, E1 0, E2 0, E3 0, E4 0}
LIN {X 518.103, Y 341.067, Z 432.88, A -110.612, B 84.801, C -94.37, E1 0, E2 0, E3 0, E4 0}
LIN {X 546.763, Y 332.708, Z 432.674, A -110.612, B 84.801, C -94.37, E1 0, E2 0, E3 0, E4 0}
LIN {X 528.89, Y 332.734, Z 433.244, A -110.612, B 84.801, C -94.37, E1 0, E2 0, E3 0, E4 0}
LIN {X 517.363, Y 336.096, Z 433.327, A -110.612, B 84.801, C -94.37, E1 0, E2 0, E3 0, E4 0}
LIN {X 583.606, Y 350.021, Z 430.02, A -110.612, B 84.801, C -94.37, E1 0, E2 0, E3 0, E4 0}
LIN {X 583.536, Y 349.837, Z 427.855, A -110.612, B 84.801, C -94.37, E1 0, E2 0, E3 0, E4 0}
LIN {X 578.97, Y 330.89, Z 429.614, A -110.612, B 84.801, C -94.37, E1 0, E2 0, E3 0, E4 0}
LIN {X 516.968, Y 332.318, Z 431.479, A -110.612, B 84.801, C -94.37, E1 0, E2 0, E3 0, E4 0}
LIN {X 514.857, Y 332.389, Z 431.54, A -110.612, B 84.801, C -94.37, E1 0, E2 0, E3 0, E4 0}
LIN {X 521.069, Y 359.585, Z 429.025, A -110.612, B 84.801, C -94.37, E1 0, E2 0, E3 0, E4 0}
LIN {X 521.076, Y 360.009, Z 428.989, A -110.612, B 84.801, C -94.37, E1 0, E2 0, E3 0, E4 0}
LIN {X 524.23, Y 368.802, Z 428.139, A -110.612, B 84.801, C -94.37, E1 0, E2 0, E3 0, E4 0}
LIN {X 526.273, Y 370.465, Z 427.932, A -110.612, B 84.801, C -94.37, E1 0, E2 0, E3 0, E4 0}
LIN {X 526.33, Y 370.561, Z 427.922, A -110.612, B 84.801, C -94.37, E1 0, E2 0, E3 0, E4 0}
LIN {X 527.658, Y 371.103, Z 427.834, A -110.612, B 84.801, C -94.37, E1 0, E2 0, E3 0, E4 0}
LIN {X 532.804, Y 370.334, Z 427.734, A -110.612, B 84.801, C -94.37, E1 0, E2 0, E3 0, E4 0}
LIN {X 533.072, Y 370.12, Z 427.744, A -110.612, B 84.801, C -94.37, E1 0, E2 0, E3 0, E4 0}
LIN {X 538.545, Y 369.112, Z 427.654, A -110.612, B 84.801, C -94.37, E1 0, E2 0, E3 0, E4 0}
LIN {X 539.294, Y 369.21, Z 427.622, A -110.612, B 84.801, C -94.37, E1 0, E2 0, E3 0, E4 0}
LIN {X 550.385, Y 367.261, Z 427.433, A -110.612, B 84.801, C -94.37, E1 0, E2 0, E3 0, E4 0}
LIN {X 550.478, Y 367.182, Z 427.437, A -110.612, B 84.801, C -94.37, E1 0, E2 0, E3 0, E4 0}
LIN {X 550.477, Y 367.17, Z 427.438, A -110.612, B 84.801, C -94.37, E1 0, E2 0, E3 0, E4 0}
LIN {X 550.54, Y 367.007, Z 427.45, A -110.612, B 84.801, C -94.37, E1 0, E2 0, E3 0, E4 0}
LIN {X 551.521, Y 365.741, Z 427.526, A -110.612, B 84.801, C -94.37, E1 0, E2 0, E3 0, E4 0}
LIN {X 557.292, Y 363.883, Z 427.499, A -110.612, B 84.801, C -94.37, E1 0, E2 0, E3 0, E4 0}
LIN {X 558.647, Y 364.028, Z 427.444, A -110.612, B 84.801, C -94.37, E1 0, E2 0, E3 0, E4 0}
LIN {X 560.958, Y 365.004, Z 427.286, A -110.612, B 84.801, C -94.37, E1 0, E2 0, E3 0, E4 0}
LIN {X 561.538, Y 365.066, Z 427.262, A -110.612, B 84.801, C -94.37, E1 0, E2 0, E3 0, E4 0}
LIN {X 579.793, Y 361.245, Z 427.003, A -110.612, B 84.801, C -94.37, E1 0, E2 0, E3 0, E4 0}
LIN {X 584.267, Y 360.582, Z 426.916, A -110.612, B 84.801, C -94.37, E1 0, E2 0, E3 0, E4 0}
LIN {X 584.527, Y 360.482, Z 426.917, A -110.612, B 84.801, C -94.37, E1 0, E2 0, E3 0, E4 0}
LIN {X 585.399, Y 359.106, Z 427.006, A -110.612, B 84.801, C -94.37, E1 0, E2 0, E3 0, E4 0}
LIN {X 585.598, Y 358.391, Z 427.06, A -110.612, B 84.801, C -94.37, E1 0, E2 0, E3 0, E4 0}
LIN {X 583.536, Y 349.837, Z 427.855, A -110.612, B 84.801, C -94.37, E1 0, E2 0, E3 0, E4 0}
LIN {X 560.507, Y 364.804, Z 427.318, A -110.612, B 84.801, C -94.37, E1 0, E2 0, E3 0, E4 0}
LIN {X 585.6, Y 357.486, Z 427.137, A -110.612, B 84.801, C -94.37, E1 0, E2 0, E3 0, E4 0}
LIN {X 584.414, Y 352.645, Z 427.587, A -110.612, B 84.801, C -94.37, E1 0, E2 0, E3 0, E4 0}
LIN {X 525.529, Y 369.819, Z 428.011, A -110.612, B 84.801, C -94.37, E1 0, E2 0, E3 0, E4 0}
LIN {X 522.763, Y 365.439, Z 428.473, A -110.612, B 84.801, C -94.37, E1 0, E2 0, E3 0, E4 0}
LIN {X 583.251, Y 347.796, Z 428.038, A -110.612, B 84.801, C -94.37, E1 0, E2 0, E3 0, E4 0}
LIN {X 582.149, Y 342.931, Z 428.487, A -110.612, B 84.801, C -94.37, E1 0, E2 0, E3 0, E4 0}
LIN {X 521.328, Y 360.67, Z 428.925, A -110.612, B 84.801, C -94.37, E1 0, E2 0, E3 0, E4 0}
LIN {X 519.9, Y 355.9, Z 429.377, A -110.612, B 84.801, C -94.37, E1 0, E2 0, E3 0, E4 0}
LIN {X 580.925, Y 338.101, Z 428.938, A -110.612, B 84.801, C -94.37, E1 0, E2 0, E3 0, E4 0}
LIN {X 579.682, Y 333.276, Z 429.389, A -110.612, B 84.801, C -94.37, E1 0, E2 0, E3 0, E4 0}
LIN {X 518.74, Y 351.051, Z 429.827, A -110.612, B 84.801, C -94.37, E1 0, E2 0, E3 0, E4 0}
LIN {X 517.721, Y 346.161, Z 430.276, A -110.612, B 84.801, C -94.37, E1 0, E2 0, E3 0, E4 0}
LIN {X 567.295, Y 331.702, Z 429.919, A -110.612, B 84.801, C -94.37, E1 0, E2 0, E3 0, E4 0}
LIN {X 546.773, Y 332.5, Z 430.509, A -110.612, B 84.801, C -94.37, E1 0, E2 0, E3 0, E4 0}
LIN {X 516.775, Y 341.25, Z 430.724, A -110.612, B 84.801, C -94.37, E1 0, E2 0, E3 0, E4 0}
LIN {X 515.501, Y 336.434, Z 431.175, A -110.612, B 84.801, C -94.37, E1 0, E2 0, E3 0, E4 0}
LIN {X 528.872, Y 332.535, Z 431.079, A -110.612, B 84.801, C -94.37, E1 0, E2 0, E3 0, E4 0}
LIN {X 585.498, Y 349.332, Z 427.835, A -110.612, B 84.801, C -94.37, E1 0, E2 0, E3 0, E4 0}
LIN {X 585.429, Y 349.148, Z 425.67, A -110.612, B 84.801, C -94.37, E1 0, E2 0, E3 0, E4 0}
LIN {X 580.677, Y 330.589, Z 427.402, A -110.612, B 84.801, C -94.37, E1 0, E2 0, E3 0, E4 0}
LIN {X 516.897, Y 332.112, Z 429.316, A -110.612, B 84.801, C -94.37, E1 0, E2 0, E3 0, E4 0}
LIN {X 513.004, Y 332.29, Z 429.425, A -110.612, B 84.801, C -94.37, E1 0, E2 0, E3 0, E4 0}
LIN {X 519.716, Y 360.243, Z 426.83, A -110.612, B 84.801, C -94.37, E1 0, E2 0, E3 0, E4 0}
LIN {X 519.726, Y 360.816, Z 426.781, A -110.612, B 84.801, C -94.37, E1 0, E2 0, E3 0, E4 0}
LIN {X 523.289, Y 370.524, Z 425.84, A -110.612, B 84.801, C -94.37, E1 0, E2 0, E3 0, E4 0}
LIN {X 525.377, Y 371.468, Z 425.693, A -110.612, B 84.801, C -94.37, E1 0, E2 0, E3 0, E4 0}
LIN {X 532.354, Y 370.433, Z 425.557, A -110.612, B 84.801, C -94.37, E1 0, E2 0, E3 0, E4 0}
LIN {X 548.253, Y 367.663, Z 425.284, A -110.612, B 84.801, C -94.37, E1 0, E2 0, E3 0, E4 0}
LIN {X 549.525, Y 367.033, Z 425.297, A -110.612, B 84.801, C -94.37, E1 0, E2 0, E3 0, E4 0}
LIN {X 550.505, Y 366.201, Z 425.336, A -110.612, B 84.801, C -94.37, E1 0, E2 0, E3 0, E4 0}
LIN {X 554.521, Y 364.993, Z 425.311, A -110.612, B 84.801, C -94.37, E1 0, E2 0, E3 0, E4 0}
LIN {X 557.225, Y 365.181, Z 425.208, A -110.612, B 84.801, C -94.37, E1 0, E2 0, E3 0, E4 0}
LIN {X 558.328, Y 364.798, Z 425.205, A -110.612, B 84.801, C -94.37, E1 0, E2 0, E3 0, E4 0}
LIN {X 558.792, Y 365.469, Z 425.133, A -110.612, B 84.801, C -94.37, E1 0, E2 0, E3 0, E4 0}
LIN {X 559.606, Y 365.564, Z 425.099, A -110.612, B 84.801, C -94.37, E1 0, E2 0, E3 0, E4 0}
LIN {X 584.421, Y 360.759, Z 424.714, A -110.612, B 84.801, C -94.37, E1 0, E2 0, E3 0, E4 0}
LIN {X 586.042, Y 360.196, Z 424.71, A -110.612, B 84.801, C -94.37, E1 0, E2 0, E3 0, E4 0}
LIN {X 586.504, Y 359.643, Z 424.742, A -110.612, B 84.801, C -94.37, E1 0, E2 0, E3 0, E4 0}
LIN {X 587.102, Y 358.312, Z 424.836, A -110.612, B 84.801, C -94.37, E1 0, E2 0, E3 0, E4 0}
LIN {X 587.349, Y 356.649, Z 424.97, A -110.612, B 84.801, C -94.37, E1 0, E2 0, E3 0, E4 0}
LIN {X 585.429, Y 349.148, Z 425.67, A -110.612, B 84.801, C -94.37, E1 0, E2 0, E3 0, E4 0}
LIN {X 587.331, Y 356.776, Z 424.959, A -110.612, B 84.801, C -94.37, E1 0, E2 0, E3 0, E4 0}
LIN {X 558.579, Y 365.162, Z 425.166, A -110.612, B 84.801, C -94.37, E1 0, E2 0, E3 0, E4 0}
LIN {X 523.134, Y 370.313, Z 425.863, A -110.612, B 84.801, C -94.37, E1 0, E2 0, E3 0, E4 0}
LIN {X 586.126, Y 351.94, Z 425.41, A -110.612, B 84.801, C -94.37, E1 0, E2 0, E3 0, E4 0}
LIN {X 584.86, Y 347.123, Z 425.861, A -110.612, B 84.801, C -94.37, E1 0, E2 0, E3 0, E4 0}
LIN {X 521.221, Y 365.684, Z 426.318, A -110.612, B 84.801, C -94.37, E1 0, E2 0, E3 0, E4 0}
LIN {X 519.757, Y 360.924, Z 426.771, A -110.612, B 84.801, C -94.37, E1 0, E2 0, E3 0, E4 0}
LIN {X 583.82, Y 342.239, Z 426.31, A -110.612, B 84.801, C -94.37, E1 0, E2 0, E3 0, E4 0}
LIN {X 582.502, Y 337.436, Z 426.761, A -110.612, B 84.801, C -94.37, E1 0, E2 0, E3 0, E4 0}
LIN {X 518.3, Y 356.162, Z 427.223, A -110.612, B 84.801, C -94.37, E1 0, E2 0, E3 0, E4 0}
LIN {X 517.173, Y 351.303, Z 427.673, A -110.612, B 84.801, C -94.37, E1 0, E2 0, E3 0, E4 0}
LIN {X 581.23, Y 332.62, Z 427.212, A -110.612, B 84.801, C -94.37, E1 0, E2 0, E3 0, E4 0}
LIN {X 567.31, Y 331.493, Z 427.754, A -110.612, B 84.801, C -94.37, E1 0, E2 0, E3 0, E4 0}
LIN {X 516.211, Y 346.397, Z 428.121, A -110.612, B 84.801, C -94.37, E1 0, E2 0, E3 0, E4 0}
LIN {X 515.15, Y 341.519, Z 428.571, A -110.612, B 84.801, C -94.37, E1 0, E2 0, E3 0, E4 0}
LIN {X 546.795, Y 332.289, Z 428.343, A -110.612, B 84.801, C -94.37, E1 0, E2 0, E3 0, E4 0}
LIN {X 528.864, Y 332.332, Z 428.914, A -110.612, B 84.801, C -94.37, E1 0, E2 0, E3 0, E4 0}
LIN {X 514.073, Y 336.646, Z 429.02, A -110.612, B 84.801, C -94.37, E1 0, E2 0, E3 0, E4 0}
LIN {X 587.339, Y 348.675, Z 425.649, A -110.612, B 84.801, C -94.37, E1 0, E2 0, E3 0, E4 0}
LIN {X 587.269, Y 348.491, Z 423.484, A -110.612, B 84.801, C -94.37, E1 0, E2 0, E3 0, E4 0}
LIN {X 582.753, Y 330.166, Z 425.189, A -110.612, B 84.801, C -94.37, E1 0, E2 0, E3 0, E4 0}
LIN {X 516.815, Y 331.927, Z 427.151, A -110.612, B 84.801, C -94.37, E1 0, E2 0, E3 0, E4 0}
LIN {X 511.417, Y 332.231, Z 427.298, A -110.612, B 84.801, C -94.37, E1 0, E2 0, E3 0, E4 0}
LIN {X 516.254, Y 351.299, Z 425.52, A -110.612, B 84.801, C -94.37, E1 0, E2 0, E3 0, E4 0}
LIN {X 516.757, Y 354.353, Z 425.243, A -110.612, B 84.801, C -94.37, E1 0, E2 0, E3 0, E4 0}
LIN {X 521.395, Y 370.335, Z 423.734, A -110.612, B 84.801, C -94.37, E1 0, E2 0, E3 0, E4 0}
LIN {X 522.393, Y 371.263, Z 423.623, A -110.612, B 84.801, C -94.37, E1 0, E2 0, E3 0, E4 0}
LIN {X 522.524, Y 371.323, Z 423.613, A -110.612, B 84.801, C -94.37, E1 0, E2 0, E3 0, E4 0}
LIN {X 524.253, Y 371.516, Z 423.542, A -110.612, B 84.801, C -94.37, E1 0, E2 0, E3 0, E4 0}
LIN {X 530.296, Y 370.816, Z 423.408, A -110.612, B 84.801, C -94.37, E1 0, E2 0, E3 0, E4 0}
LIN {X 531.745, Y 369.924, Z 423.437, A -110.612, B 84.801, C -94.37, E1 0, E2 0, E3 0, E4 0}
LIN {X 531.992, Y 369.912, Z 423.43, A -110.612, B 84.801, C -94.37, E1 0, E2 0, E3 0, E4 0}
LIN {X 532.925, Y 370.249, Z 423.372, A -110.612, B 84.801, C -94.37, E1 0, E2 0, E3 0, E4 0}
LIN {X 548.565, Y 367.444, Z 423.11, A -110.612, B 84.801, C -94.37, E1 0, E2 0, E3 0, E4 0}
LIN {X 548.807, Y 367.23, Z 423.12, A -110.612, B 84.801, C -94.37, E1 0, E2 0, E3 0, E4 0}
LIN {X 549.2, Y 367.056, Z 423.122, A -110.612, B 84.801, C -94.37, E1 0, E2 0, E3 0, E4 0}
LIN {X 549.808, Y 366.562, Z 423.145, A -110.612, B 84.801, C -94.37, E1 0, E2 0, E3 0, E4 0}
LIN {X 556.818, Y 365.866, Z 422.98, A -110.612, B 84.801, C -94.37, E1 0, E2 0, E3 0, E4 0}
LIN {X 558.959, Y 365.602, Z 422.934, A -110.612, B 84.801, C -94.37, E1 0, E2 0, E3 0, E4 0}
LIN {X 559.885, Y 365.124, Z 422.945, A -110.612, B 84.801, C -94.37, E1 0, E2 0, E3 0, E4 0}
LIN {X 568.219, Y 363.81, Z 422.79, A -110.612, B 84.801, C -94.37, E1 0, E2 0, E3 0, E4 0}
LIN {X 568.558, Y 363.631, Z 422.794, A -110.612, B 84.801, C -94.37, E1 0, E2 0, E3 0, E4 0}
LIN {X 586.498, Y 360.444, Z 422.491, A -110.612, B 84.801, C -94.37, E1 0, E2 0, E3 0, E4 0}
LIN {X 587.768, Y 359.658, Z 422.517, A -110.612, B 84.801, C -94.37, E1 0, E2 0, E3 0, E4 0}
LIN {X 588.797, Y 358.186, Z 422.609, A -110.612, B 84.801, C -94.37, E1 0, E2 0, E3 0, E4 0}
LIN {X 589.057, Y 355.747, Z 422.809, A -110.612, B 84.801, C -94.37, E1 0, E2 0, E3 0, E4 0}
LIN {X 587.269, Y 348.491, Z 423.484, A -110.612, B 84.801, C -94.37, E1 0, E2 0, E3 0, E4 0}
LIN {X 555.764, Y 365.778, Z 423.021, A -110.612, B 84.801, C -94.37, E1 0, E2 0, E3 0, E4 0}
LIN {X 589.011, Y 356.081, Z 422.782, A -110.612, B 84.801, C -94.37, E1 0, E2 0, E3 0, E4 0}
LIN {X 587.7, Y 351.277, Z 423.233, A -110.612, B 84.801, C -94.37, E1 0, E2 0, E3 0, E4 0}
LIN {X 521.625, Y 370.548, Z 423.708, A -110.612, B 84.801, C -94.37, E1 0, E2 0, E3 0, E4 0}
LIN {X 519.881, Y 365.87, Z 424.163, A -110.612, B 84.801, C -94.37, E1 0, E2 0, E3 0, E4 0}
LIN {X 586.204, Y 346.526, Z 423.686, A -110.612, B 84.801, C -94.37, E1 0, E2 0, E3 0, E4 0}
LIN {X 584.986, Y 341.694, Z 424.136, A -110.612, B 84.801, C -94.37, E1 0, E2 0, E3 0, E4 0}
LIN {X 518.482, Y 361.091, Z 424.614, A -110.612, B 84.801, C -94.37, E1 0, E2 0, E3 0, E4 0}
LIN {X 517.199, Y 356.278, Z 425.065, A -110.612, B 84.801, C -94.37, E1 0, E2 0, E3 0, E4 0}
LIN {X 584.056, Y 336.779, Z 424.584, A -110.612, B 84.801, C -94.37, E1 0, E2 0, E3 0, E4 0}
LIN {X 583.256, Y 331.825, Z 425.032, A -110.612, B 84.801, C -94.37, E1 0, E2 0, E3 0, E4 0}
LIN {X 516.269, Y 351.362, Z 425.514, A -110.612, B 84.801, C -94.37, E1 0, E2 0, E3 0, E4 0}
LIN {X 514.87, Y 346.583, Z 425.965, A -110.612, B 84.801, C -94.37, E1 0, E2 0, E3 0, E4 0}
LIN {X 567.242, Y 331.309, Z 425.589, A -110.612, B 84.801, C -94.37, E1 0, E2 0, E3 0, E4 0}
LIN {X 546.728, Y 332.105, Z 426.178, A -110.612, B 84.801, C -94.37, E1 0, E2 0, E3 0, E4 0}
LIN {X 513.756, Y 341.721, Z 426.415, A -110.612, B 84.801, C -94.37, E1 0, E2 0, E3 0, E4 0}
LIN {X 512.754, Y 336.826, Z 426.864, A -110.612, B 84.801, C -94.37, E1 0, E2 0, E3 0, E4 0}
LIN {X 528.791, Y 332.149, Z 426.749, A -110.612, B 84.801, C -94.37, E1 0, E2 0, E3 0, E4 0}
LIN {X 588.688, Y 348.121, Z 423.47, A -110.612, B 84.801, C -94.37, E1 0, E2 0, E3 0, E4 0}
LIN {X 588.619, Y 347.937, Z 421.305, A -110.612, B 84.801, C -94.37, E1 0, E2 0, E3 0, E4 0}
LIN {X 583.926, Y 329.877, Z 422.993, A -110.612, B 84.801, C -94.37, E1 0, E2 0, E3 0, E4 0}
LIN {X 516.719, Y 331.727, Z 424.988, A -110.612, B 84.801, C -94.37, E1 0, E2 0, E3 0, E4 0}
LIN {X 510.112, Y 332.131, Z 425.166, A -110.612, B 84.801, C -94.37, E1 0, E2 0, E3 0, E4 0}
LIN {X 514.64, Y 349.657, Z 423.528, A -110.612, B 84.801, C -94.37, E1 0, E2 0, E3 0, E4 0}
LIN {X 515.304, Y 351.535, Z 423.347, A -110.612, B 84.801, C -94.37, E1 0, E2 0, E3 0, E4 0}
LIN {X 516.255, Y 355.818, Z 422.952, A -110.612, B 84.801, C -94.37, E1 0, E2 0, E3 0, E4 0}
LIN {X 516.204, Y 355.822, Z 422.953, A -110.612, B 84.801, C -94.37, E1 0, E2 0, E3 0, E4 0}
LIN {X 520.03, Y 370.88, Z 421.548, A -110.612, B 84.801, C -94.37, E1 0, E2 0, E3 0, E4 0}
LIN {X 521.427, Y 371.611, Z 421.441, A -110.612, B 84.801, C -94.37, E1 0, E2 0, E3 0, E4 0}
LIN {X 522.738, Y 371.763, Z 421.386, A -110.612, B 84.801, C -94.37, E1 0, E2 0, E3 0, E4 0}
LIN {X 523.423, Y 371.567, Z 421.381, A -110.612, B 84.801, C -94.37, E1 0, E2 0, E3 0, E4 0}
LIN {X 524.907, Y 371.578, Z 421.333, A -110.612, B 84.801, C -94.37, E1 0, E2 0, E3 0, E4 0}
LIN {X 527.12, Y 371.311, Z 421.284, A -110.612, B 84.801, C -94.37, E1 0, E2 0, E3 0, E4 0}
LIN {X 527.868, Y 370.715, Z 421.311, A -110.612, B 84.801, C -94.37, E1 0, E2 0, E3 0, E4 0}
LIN {X 530.313, Y 370.445, Z 421.256, A -110.612, B 84.801, C -94.37, E1 0, E2 0, E3 0, E4 0}
LIN {X 530.399, Y 370.555, Z 421.244, A -110.612, B 84.801, C -94.37, E1 0, E2 0, E3 0, E4 0}
LIN {X 532.275, Y 370.415, Z 421.196, A -110.612, B 84.801, C -94.37, E1 0, E2 0, E3 0, E4 0}
LIN {X 532.93, Y 370.038, Z 421.207, A -110.612, B 84.801, C -94.37, E1 0, E2 0, E3 0, E4 0}
LIN {X 533.565, Y 369.897, Z 421.198, A -110.612, B 84.801, C -94.37, E1 0, E2 0, E3 0, E4 0}
LIN {X 534.415, Y 370.011, Z 421.161, A -110.612, B 84.801, C -94.37, E1 0, E2 0, E3 0, E4 0}
LIN {X 546.141, Y 368.047, Z 420.953, A -110.612, B 84.801, C -94.37, E1 0, E2 0, E3 0, E4 0}
LIN {X 548.572, Y 366.223, Z 421.031, A -110.612, B 84.801, C -94.37, E1 0, E2 0, E3 0, E4 0}
LIN {X 549.627, Y 366.475, Z 420.975, A -110.612, B 84.801, C -94.37, E1 0, E2 0, E3 0, E4 0}
LIN {X 552.782, Y 365.995, Z 420.915, A -110.612, B 84.801, C -94.37, E1 0, E2 0, E3 0, E4 0}
LIN {X 554.913, Y 366.351, Z 420.817, A -110.612, B 84.801, C -94.37, E1 0, E2 0, E3 0, E4 0}
LIN {X 564.484, Y 364.414, Z 420.675, A -110.612, B 84.801, C -94.37, E1 0, E2 0, E3 0, E4 0}
LIN {X 565.781, Y 363.738, Z 420.691, A -110.612, B 84.801, C -94.37, E1 0, E2 0, E3 0, E4 0}
LIN {X 565.989, Y 363.697, Z 420.688, A -110.612, B 84.801, C -94.37, E1 0, E2 0, E3 0, E4 0}
LIN {X 566.915, Y 363.919, Z 420.639, A -110.612, B 84.801, C -94.37, E1 0, E2 0, E3 0, E4 0}
LIN {X 573.459, Y 362.748, Z 420.529, A -110.612, B 84.801, C -94.37, E1 0, E2 0, E3 0, E4 0}
LIN {X 574.202, Y 362.267, Z 420.546, A -110.612, B 84.801, C -94.37, E1 0, E2 0, E3 0, E4 0}
LIN {X 588.729, Y 360.063, Z 420.269, A -110.612, B 84.801, C -94.37, E1 0, E2 0, E3 0, E4 0}
LIN {X 589.845, Y 359.516, Z 420.28, A -110.612, B 84.801, C -94.37, E1 0, E2 0, E3 0, E4 0}
LIN {X 589.949, Y 359.403, Z 420.286, A -110.612, B 84.801, C -94.37, E1 0, E2 0, E3 0, E4 0}
LIN {X 590.763, Y 356.186, Z 420.534, A -110.612, B 84.801, C -94.37, E1 0, E2 0, E3 0, E4 0}
LIN {X 588.619, Y 347.937, Z 421.305, A -110.612, B 84.801, C -94.37, E1 0, E2 0, E3 0, E4 0}
LIN {X 553.761, Y 366.158, Z 420.87, A -110.612, B 84.801, C -94.37, E1 0, E2 0, E3 0, E4 0}
LIN {X 590.695, Y 355.386, Z 420.604, A -110.612, B 84.801, C -94.37, E1 0, E2 0, E3 0, E4 0}
LIN {X 589.228, Y 350.627, Z 421.056, A -110.612, B 84.801, C -94.37, E1 0, E2 0, E3 0, E4 0}
LIN {X 520.009, Y 370.815, Z 421.554, A -110.612, B 84.801, C -94.37, E1 0, E2 0, E3 0, E4 0}
LIN {X 518.731, Y 366.001, Z 422.005, A -110.612, B 84.801, C -94.37, E1 0, E2 0, E3 0, E4 0}
LIN {X 587.548, Y 345.93, Z 421.51, A -110.612, B 84.801, C -94.37, E1 0, E2 0, E3 0, E4 0}
LIN {X 586.024, Y 341.187, Z 421.963, A -110.612, B 84.801, C -94.37, E1 0, E2 0, E3 0, E4 0}
LIN {X 517.512, Y 361.169, Z 422.456, A -110.612, B 84.801, C -94.37, E1 0, E2 0, E3 0, E4 0}
LIN {X 516.338, Y 356.324, Z 422.906, A -110.612, B 84.801, C -94.37, E1 0, E2 0, E3 0, E4 0}
LIN {X 584.869, Y 336.337, Z 422.413, A -110.612, B 84.801, C -94.37, E1 0, E2 0, E3 0, E4 0}
LIN {X 584.263, Y 331.326, Z 422.859, A -110.612, B 84.801, C -94.37, E1 0, E2 0, E3 0, E4 0}
LIN {X 515.26, Y 351.452, Z 423.355, A -110.612, B 84.801, C -94.37, E1 0, E2 0, E3 0, E4 0}
LIN {X 513.944, Y 346.649, Z 423.806, A -110.612, B 84.801, C -94.37, E1 0, E2 0, E3 0, E4 0}
LIN {X 567.24, Y 331.104, Z 423.423, A -110.612, B 84.801, C -94.37, E1 0, E2 0, E3 0, E4 0}
LIN {X 546.734, Y 331.898, Z 424.013, A -110.612, B 84.801, C -94.37, E1 0, E2 0, E3 0, E4 0}
LIN {X 512.57, Y 341.862, Z 424.258, A -110.612, B 84.801, C -94.37, E1 0, E2 0, E3 0, E4 0}
LIN {X 511.41, Y 337.014, Z 424.708, A -110.612, B 84.801, C -94.37, E1 0, E2 0, E3 0, E4 0}
LIN {X 528.764, Y 331.952, Z 424.583, A -110.612, B 84.801, C -94.37, E1 0, E2 0, E3 0, E4 0}
LIN {X 510.469, Y 332.101, Z 425.157, A -110.612, B 84.801, C -94.37, E1 0, E2 0, E3 0, E4 0}
LIN {X 510.134, Y 332.199, Z 425.159, A -110.612, B 84.801, C -94.37, E1 0, E2 0, E3 0, E4 0}
LIN {X 589.728, Y 347.562, Z 421.301, A -110.612, B 84.801, C -94.37, E1 0, E2 0, E3 0, E4 0}
LIN {X 589.659, Y 347.378, Z 419.137, A -110.612, B 84.801, C -94.37, E1 0, E2 0, E3 0, E4 0}
LIN {X 587.097, Y 339.783, Z 419.865, A -110.612, B 84.801, C -94.37, E1 0, E2 0, E3 0, E4 0}
LIN {X 585.214, Y 329.63, Z 420.79, A -110.612, B 84.801, C -94.37, E1 0, E2 0, E3 0, E4 0}
LIN {X 509.74, Y 331.959, Z 423.009, A -110.612, B 84.801, C -94.37, E1 0, E2 0, E3 0, E4 0}
LIN {X 508.734, Y 332.044, Z 423.034, A -110.612, B 84.801, C -94.37, E1 0, E2 0, E3 0, E4 0}
LIN {X 515.63, Y 357.273, Z 420.665, A -110.612, B 84.801, C -94.37, E1 0, E2 0, E3 0, E4 0}
LIN {X 516.064, Y 357.812, Z 420.605, A -110.612, B 84.801, C -94.37, E1 0, E2 0, E3 0, E4 0}
LIN {X 518.001, Y 369.293, Z 419.565, A -110.612, B 84.801, C -94.37, E1 0, E2 0, E3 0, E4 0}
LIN {X 518.942, Y 371.346, Z 419.36, A -110.612, B 84.801, C -94.37, E1 0, E2 0, E3 0, E4 0}
LIN {X 519.863, Y 371.732, Z 419.298, A -110.612, B 84.801, C -94.37, E1 0, E2 0, E3 0, E4 0}
LIN {X 524.65, Y 371.688, Z 419.148, A -110.612, B 84.801, C -94.37, E1 0, E2 0, E3 0, E4 0}
LIN {X 527.44, Y 370.27, Z 419.18, A -110.612, B 84.801, C -94.37, E1 0, E2 0, E3 0, E4 0}
LIN {X 528.814, Y 370.028, Z 419.156, A -110.612, B 84.801, C -94.37, E1 0, E2 0, E3 0, E4 0}
LIN {X 529.647, Y 370.532, Z 419.087, A -110.612, B 84.801, C -94.37, E1 0, E2 0, E3 0, E4 0}
LIN {X 530.327, Y 370.563, Z 419.062, A -110.612, B 84.801, C -94.37, E1 0, E2 0, E3 0, E4 0}
LIN {X 530.399, Y 370.654, Z 419.052, A -110.612, B 84.801, C -94.37, E1 0, E2 0, E3 0, E4 0}
LIN {X 534.08, Y 369.71, Z 419.015, A -110.612, B 84.801, C -94.37, E1 0, E2 0, E3 0, E4 0}
LIN {X 535.454, Y 369.754, Z 418.967, A -110.612, B 84.801, C -94.37, E1 0, E2 0, E3 0, E4 0}
LIN {X 538.216, Y 368.744, Z 418.965, A -110.612, B 84.801, C -94.37, E1 0, E2 0, E3 0, E4 0}
LIN {X 539.877, Y 368.857, Z 418.902, A -110.612, B 84.801, C -94.37, E1 0, E2 0, E3 0, E4 0}
LIN {X 540.612, Y 368.479, Z 418.91, A -110.612, B 84.801, C -94.37, E1 0, E2 0, E3 0, E4 0}
LIN {X 541.951, Y 368.379, Z 418.876, A -110.612, B 84.801, C -94.37, E1 0, E2 0, E3 0, E4 0}
LIN {X 543.537, Y 367.744, Z 418.879, A -110.612, B 84.801, C -94.37, E1 0, E2 0, E3 0, E4 0}
LIN {X 544.139, Y 367.204, Z 418.906, A -110.612, B 84.801, C -94.37, E1 0, E2 0, E3 0, E4 0}
LIN {X 547.036, Y 366.476, Z 418.875, A -110.612, B 84.801, C -94.37, E1 0, E2 0, E3 0, E4 0}
LIN {X 547.668, Y 366.618, Z 418.843, A -110.612, B 84.801, C -94.37, E1 0, E2 0, E3 0, E4 0}
LIN {X 548.364, Y 366.574, Z 418.824, A -110.612, B 84.801, C -94.37, E1 0, E2 0, E3 0, E4 0}
LIN {X 549.131, Y 366.299, Z 418.823, A -110.612, B 84.801, C -94.37, E1 0, E2 0, E3 0, E4 0}
LIN {X 552.073, Y 366.202, Z 418.737, A -110.612, B 84.801, C -94.37, E1 0, E2 0, E3 0, E4 0}
LIN {X 552.505, Y 366.283, Z 418.717, A -110.612, B 84.801, C -94.37, E1 0, E2 0, E3 0, E4 0}
LIN {X 567.134, Y 363.855, Z 418.455, A -110.612, B 84.801, C -94.37, E1 0, E2 0, E3 0, E4 0}
LIN {X 567.378, Y 363.669, Z 418.463, A -110.612, B 84.801, C -94.37, E1 0, E2 0, E3 0, E4 0}
LIN {X 578.625, Y 361.775, Z 418.264, A -110.612, B 84.801, C -94.37, E1 0, E2 0, E3 0, E4 0}
LIN {X 578.856, Y 361.799, Z 418.255, A -110.612, B 84.801, C -94.37, E1 0, E2 0, E3 0, E4 0}
LIN {X 591.493, Y 358.908, Z 418.096, A -110.612, B 84.801, C -94.37, E1 0, E2 0, E3 0, E4 0}
LIN {X 591.885, Y 358.617, Z 418.108, A -110.612, B 84.801, C -94.37, E1 0, E2 0, E3 0, E4 0}
LIN {X 592.065, Y 358.292, Z 418.13, A -110.612, B 84.801, C -94.37, E1 0, E2 0, E3 0, E4 0}
LIN {X 592.306, Y 355.226, Z 418.383, A -110.612, B 84.801, C -94.37, E1 0, E2 0, E3 0, E4 0}
LIN {X 589.659, Y 347.378, Z 419.137, A -110.612, B 84.801, C -94.37, E1 0, E2 0, E3 0, E4 0}
LIN {X 552.857, Y 366.217, Z 418.711, A -110.612, B 84.801, C -94.37, E1 0, E2 0, E3 0, E4 0}
LIN {X 592.136, Y 354.761, Z 418.428, A -110.612, B 84.801, C -94.37, E1 0, E2 0, E3 0, E4 0}
LIN {X 590.642, Y 350.009, Z 418.881, A -110.612, B 84.801, C -94.37, E1 0, E2 0, E3 0, E4 0}
LIN {X 518.742, Y 370.98, Z 419.398, A -110.612, B 84.801, C -94.37, E1 0, E2 0, E3 0, E4 0}
LIN {X 517.598, Y 366.127, Z 419.848, A -110.612, B 84.801, C -94.37, E1 0, E2 0, E3 0, E4 0}
LIN {X 588.889, Y 345.334, Z 419.335, A -110.612, B 84.801, C -94.37, E1 0, E2 0, E3 0, E4 0}
LIN {X 587.367, Y 340.591, Z 419.788, A -110.612, B 84.801, C -94.37, E1 0, E2 0, E3 0, E4 0}
LIN {X 516.578, Y 361.237, Z 420.297, A -110.612, B 84.801, C -94.37, E1 0, E2 0, E3 0, E4 0}
LIN {X 515.325, Y 356.415, Z 420.748, A -110.612, B 84.801, C -94.37, E1 0, E2 0, E3 0, E4 0}
LIN {X 586.011, Y 335.799, Z 420.239, A -110.612, B 84.801, C -94.37, E1 0, E2 0, E3 0, E4 0}
LIN {X 585.368, Y 330.8, Z 420.686, A -110.612, B 84.801, C -94.37, E1 0, E2 0, E3 0, E4 0}
LIN {X 513.956, Y 351.628, Z 421.199, A -110.612, B 84.801, C -94.37, E1 0, E2 0, E3 0, E4 0}
LIN {X 512.647, Y 346.822, Z 421.651, A -110.612, B 84.801, C -94.37, E1 0, E2 0, E3 0, E4 0}
LIN {X 567.238, Y 330.9, Z 421.258, A -110.612, B 84.801, C -94.37, E1 0, E2 0, E3 0, E4 0}
LIN {X 546.738, Y 331.693, Z 421.847, A -110.612, B 84.801, C -94.37, E1 0, E2 0, E3 0, E4 0}
LIN {X 511.345, Y 342.015, Z 422.102, A -110.612, B 84.801, C -94.37, E1 0, E2 0, E3 0, E4 0}
LIN {X 510.226, Y 337.154, Z 422.551, A -110.612, B 84.801, C -94.37, E1 0, E2 0, E3 0, E4 0}
LIN {X 528.74, Y 331.755, Z 422.418, A -110.612, B 84.801, C -94.37, E1 0, E2 0, E3 0, E4 0}
LIN {X 510.485, Y 331.892, Z 422.991, A -110.612, B 84.801, C -94.37, E1 0, E2 0, E3 0, E4 0}
LIN {X 508.837, Y 332.373, Z 423.003, A -110.612, B 84.801, C -94.37, E1 0, E2 0, E3 0, E4 0}
LIN {X 590.932, Y 346.967, Z 419.131, A -110.612, B 84.801, C -94.37, E1 0, E2 0, E3 0, E4 0}
LIN {X 590.863, Y 346.783, Z 416.966, A -110.612, B 84.801, C -94.37, E1 0, E2 0, E3 0, E4 0}
LIN {X 588.396, Y 339.125, Z 417.697, A -110.612, B 84.801, C -94.37, E1 0, E2 0, E3 0, E4 0}
LIN {X 586.484, Y 329.398, Z 418.587, A -110.612, B 84.801, C -94.37, E1 0, E2 0, E3 0, E4 0}
LIN {X 509.648, Y 331.76, Z 420.846, A -110.612, B 84.801, C -94.37, E1 0, E2 0, E3 0, E4 0}
LIN {X 507.304, Y 331.968, Z 420.904, A -110.612, B 84.801, C -94.37, E1 0, E2 0, E3 0, E4 0}
LIN {X 517.931, Y 371.15, Z 417.227, A -110.612, B 84.801, C -94.37, E1 0, E2 0, E3 0, E4 0}
LIN {X 518.364, Y 371.576, Z 417.176, A -110.612, B 84.801, C -94.37, E1 0, E2 0, E3 0, E4 0}
LIN {X 519.478, Y 371.8, Z 417.122, A -110.612, B 84.801, C -94.37, E1 0, E2 0, E3 0, E4 0}
LIN {X 519.585, Y 371.737, Z 417.124, A -110.612, B 84.801, C -94.37, E1 0, E2 0, E3 0, E4 0}
LIN {X 519.656, Y 371.805, Z 417.116, A -110.612, B 84.801, C -94.37, E1 0, E2 0, E3 0, E4 0}
LIN {X 520.512, Y 372.066, Z 417.066, A -110.612, B 84.801, C -94.37, E1 0, E2 0, E3 0, E4 0}
LIN {X 540.232, Y 368.834, Z 416.71, A -110.612, B 84.801, C -94.37, E1 0, E2 0, E3 0, E4 0}
LIN {X 541.223, Y 367.761, Z 416.769, A -110.612, B 84.801, C -94.37, E1 0, E2 0, E3 0, E4 0}
LIN {X 553.672, Y 365.952, Z 416.524, A -110.612, B 84.801, C -94.37, E1 0, E2 0, E3 0, E4 0}
LIN {X 554.674, Y 366.095, Z 416.48, A -110.612, B 84.801, C -94.37, E1 0, E2 0, E3 0, E4 0}
LIN {X 562.188, Y 365.126, Z 416.322, A -110.612, B 84.801, C -94.37, E1 0, E2 0, E3 0, E4 0}
LIN {X 568.304, Y 363.13, Z 416.296, A -110.612, B 84.801, C -94.37, E1 0, E2 0, E3 0, E4 0}
LIN {X 577.727, Y 361.667, Z 416.119, A -110.612, B 84.801, C -94.37, E1 0, E2 0, E3 0, E4 0}
LIN {X 578.182, Y 361.714, Z 416.1, A -110.612, B 84.801, C -94.37, E1 0, E2 0, E3 0, E4 0}
LIN {X 589.577, Y 359.173, Z 415.952, A -110.612, B 84.801, C -94.37, E1 0, E2 0, E3 0, E4 0}
LIN {X 593.185, Y 358.649, Z 415.881, A -110.612, B 84.801, C -94.37, E1 0, E2 0, E3 0, E4 0}
LIN {X 594.03, Y 358.007, Z 415.909, A -110.612, B 84.801, C -94.37, E1 0, E2 0, E3 0, E4 0}
LIN {X 594.04, Y 356.645, Z 416.024, A -110.612, B 84.801, C -94.37, E1 0, E2 0, E3 0, E4 0}
LIN {X 590.863, Y 346.783, Z 416.966, A -110.612, B 84.801, C -94.37, E1 0, E2 0, E3 0, E4 0}
LIN {X 552.539, Y 366.105, Z 416.548, A -110.612, B 84.801, C -94.37, E1 0, E2 0, E3 0, E4 0}
LIN {X 593.359, Y 354.2, Z 416.254, A -110.612, B 84.801, C -94.37, E1 0, E2 0, E3 0, E4 0}
LIN {X 592.023, Y 349.402, Z 416.706, A -110.612, B 84.801, C -94.37, E1 0, E2 0, E3 0, E4 0}
LIN {X 517.881, Y 371.027, Z 417.239, A -110.612, B 84.801, C -94.37, E1 0, E2 0, E3 0, E4 0}
LIN {X 516.358, Y 366.284, Z 417.691, A -110.612, B 84.801, C -94.37, E1 0, E2 0, E3 0, E4 0}
LIN {X 590.217, Y 344.742, Z 417.16, A -110.612, B 84.801, C -94.37, E1 0, E2 0, E3 0, E4 0}
LIN {X 588.756, Y 339.981, Z 417.612, A -110.612, B 84.801, C -94.37, E1 0, E2 0, E3 0, E4 0}
LIN {X 515.373, Y 361.384, Z 418.14, A -110.612, B 84.801, C -94.37, E1 0, E2 0, E3 0, E4 0}
LIN {X 513.91, Y 356.624, Z 418.592, A -110.612, B 84.801, C -94.37, E1 0, E2 0, E3 0, E4 0}
LIN {X 587.433, Y 335.18, Z 418.064, A -110.612, B 84.801, C -94.37, E1 0, E2 0, E3 0, E4 0}
LIN {X 586.59, Y 330.239, Z 418.512, A -110.612, B 84.801, C -94.37, E1 0, E2 0, E3 0, E4 0}
LIN {X 512.808, Y 351.758, Z 419.042, A -110.612, B 84.801, C -94.37, E1 0, E2 0, E3 0, E4 0}
LIN {X 511.535, Y 346.942, Z 419.493, A -110.612, B 84.801, C -94.37, E1 0, E2 0, E3 0, E4 0}
LIN {X 567.23, Y 330.698, Z 419.093, A -110.612, B 84.801, C -94.37, E1 0, E2 0, E3 0, E4 0}
LIN {X 546.736, Y 331.489, Z 419.682, A -110.612, B 84.801, C -94.37, E1 0, E2 0, E3 0, E4 0}
LIN {X 510.218, Y 342.139, Z 419.944, A -110.612, B 84.801, C -94.37, E1 0, E2 0, E3 0, E4 0}
LIN {X 508.801, Y 337.365, Z 420.396, A -110.612, B 84.801, C -94.37, E1 0, E2 0, E3 0, E4 0}
LIN {X 528.709, Y 331.559, Z 420.253, A -110.612, B 84.801, C -94.37, E1 0, E2 0, E3 0, E4 0}
LIN {X 510.496, Y 331.684, Z 420.826, A -110.612, B 84.801, C -94.37, E1 0, E2 0, E3 0, E4 0}
LIN {X 507.498, Y 332.558, Z 420.847, A -110.612, B 84.801, C -94.37, E1 0, E2 0, E3 0, E4 0}
LIN {X 592.264, Y 346.357, Z 416.957, A -110.612, B 84.801, C -94.37, E1 0, E2 0, E3 0, E4 0}
LIN {X 592.195, Y 346.173, Z 414.792, A -110.612, B 84.801, C -94.37, E1 0, E2 0, E3 0, E4 0}
LIN {X 591.503, Y 343.888, Z 415.009, A -110.612, B 84.801, C -94.37, E1 0, E2 0, E3 0, E4 0}
LIN {X 587.502, Y 329.207, Z 416.387, A -110.612, B 84.801, C -94.37, E1 0, E2 0, E3 0, E4 0}
LIN {X 509.363, Y 331.565, Z 418.689, A -110.612, B 84.801, C -94.37, E1 0, E2 0, E3 0, E4 0}
LIN {X 506.196, Y 331.869, Z 418.764, A -110.612, B 84.801, C -94.37, E1 0, E2 0, E3 0, E4 0}
LIN {X 516.633, Y 370.893, Z 415.107, A -110.612, B 84.801, C -94.37, E1 0, E2 0, E3 0, E4 0}
LIN {X 517.946, Y 372.184, Z 414.955, A -110.612, B 84.801, C -94.37, E1 0, E2 0, E3 0, E4 0}
LIN {X 518.821, Y 372.38, Z 414.91, A -110.612, B 84.801, C -94.37, E1 0, E2 0, E3 0, E4 0}
LIN {X 530.533, Y 370.387, Z 414.705, A -110.612, B 84.801, C -94.37, E1 0, E2 0, E3 0, E4 0}
LIN {X 531.924, Y 370.307, Z 414.667, A -110.612, B 84.801, C -94.37, E1 0, E2 0, E3 0, E4 0}
LIN {X 540.854, Y 368.719, Z 414.516, A -110.612, B 84.801, C -94.37, E1 0, E2 0, E3 0, E4 0}
LIN {X 543.253, Y 367.523, Z 414.541, A -110.612, B 84.801, C -94.37, E1 0, E2 0, E3 0, E4 0}
LIN {X 543.546, Y 367.563, Z 414.529, A -110.612, B 84.801, C -94.37, E1 0, E2 0, E3 0, E4 0}
LIN {X 543.971, Y 367.854, Z 414.49, A -110.612, B 84.801, C -94.37, E1 0, E2 0, E3 0, E4 0}
LIN {X 544.993, Y 368.036, Z 414.442, A -110.612, B 84.801, C -94.37, E1 0, E2 0, E3 0, E4 0}
LIN {X 548.694, Y 367.359, Z 414.381, A -110.612, B 84.801, C -94.37, E1 0, E2 0, E3 0, E4 0}
LIN {X 549.456, Y 366.439, Z 414.435, A -110.612, B 84.801, C -94.37, E1 0, E2 0, E3 0, E4 0}
LIN {X 551.312, Y 365.856, Z 414.425, A -110.612, B 84.801, C -94.37, E1 0, E2 0, E3 0, E4 0}
LIN {X 562.244, Y 365.231, Z 414.128, A -110.612, B 84.801, C -94.37, E1 0, E2 0, E3 0, E4 0}
LIN {X 564.023, Y 364.71, Z 414.116, A -110.612, B 84.801, C -94.37, E1 0, E2 0, E3 0, E4 0}
LIN {X 565.517, Y 363.498, Z 414.171, A -110.612, B 84.801, C -94.37, E1 0, E2 0, E3 0, E4 0}
LIN {X 576.596, Y 361.104, Z 414.02, A -110.612, B 84.801, C -94.37, E1 0, E2 0, E3 0, E4 0}
LIN {X 578.474, Y 360.831, Z 413.983, A -110.612, B 84.801, C -94.37, E1 0, E2 0, E3 0, E4 0}
LIN {X 579.278, Y 360.608, Z 413.976, A -110.612, B 84.801, C -94.37, E1 0, E2 0, E3 0, E4 0}
LIN {X 581.471, Y 361.134, Z 413.861, A -110.612, B 84.801, C -94.37, E1 0, E2 0, E3 0, E4 0}
LIN {X 595.014, Y 357.676, Z 413.722, A -110.612, B 84.801, C -94.37, E1 0, E2 0, E3 0, E4 0}
LIN {X 595.125, Y 357.727, Z 413.714, A -110.612, B 84.801, C -94.37, E1 0, E2 0, E3 0, E4 0}
LIN {X 595.232, Y 357.666, Z 413.716, A -110.612, B 84.801, C -94.37, E1 0, E2 0, E3 0, E4 0}
LIN {X 595.352, Y 357.483, Z 413.728, A -110.612, B 84.801, C -94.37, E1 0, E2 0, E3 0, E4 0}
LIN {X 595.578, Y 357.341, Z 413.732, A -110.612, B 84.801, C -94.37, E1 0, E2 0, E3 0, E4 0}
LIN {X 592.195, Y 346.173, Z 414.792, A -110.612, B 84.801, C -94.37, E1 0, E2 0, E3 0, E4 0}
LIN {X 594.684, Y 353.609, Z 414.079, A -110.612, B 84.801, C -94.37, E1 0, E2 0, E3 0, E4 0}
LIN {X 553.923, Y 365.497, Z 414.372, A -110.612, B 84.801, C -94.37, E1 0, E2 0, E3 0, E4 0}
LIN {X 545.227, Y 368.033, Z 414.435, A -110.612, B 84.801, C -94.37, E1 0, E2 0, E3 0, E4 0}
LIN {X 549.101, Y 366.903, Z 414.407, A -110.612, B 84.801, C -94.37, E1 0, E2 0, E3 0, E4 0}
LIN {X 593.422, Y 348.79, Z 414.53, A -110.612, B 84.801, C -94.37, E1 0, E2 0, E3 0, E4 0}
LIN {X 516.863, Y 371.119, Z 415.08, A -110.612, B 84.801, C -94.37, E1 0, E2 0, E3 0, E4 0}
LIN {X 515.434, Y 366.349, Z 415.532, A -110.612, B 84.801, C -94.37, E1 0, E2 0, E3 0, E4 0}
LIN {X 591.641, Y 344.122, Z 414.984, A -110.612, B 84.801, C -94.37, E1 0, E2 0, E3 0, E4 0}
LIN {X 590.145, Y 339.371, Z 415.437, A -110.612, B 84.801, C -94.37, E1 0, E2 0, E3 0, E4 0}
LIN {X 514.282, Y 361.497, Z 415.982, A -110.612, B 84.801, C -94.37, E1 0, E2 0, E3 0, E4 0}
LIN {X 512.939, Y 356.702, Z 416.434, A -110.612, B 84.801, C -94.37, E1 0, E2 0, E3 0, E4 0}
LIN {X 588.866, Y 334.557, Z 415.888, A -110.612, B 84.801, C -94.37, E1 0, E2 0, E3 0, E4 0}
LIN {X 587.622, Y 329.733, Z 416.338, A -110.612, B 84.801, C -94.37, E1 0, E2 0, E3 0, E4 0}
LIN {X 511.579, Y 351.912, Z 416.885, A -110.612, B 84.801, C -94.37, E1 0, E2 0, E3 0, E4 0}
LIN {X 510.509, Y 347.037, Z 417.335, A -110.612, B 84.801, C -94.37, E1 0, E2 0, E3 0, E4 0}
LIN {X 567.244, Y 330.489, Z 416.927, A -110.612, B 84.801, C -94.37, E1 0, E2 0, E3 0, E4 0}
LIN {X 546.745, Y 331.281, Z 417.516, A -110.612, B 84.801, C -94.37, E1 0, E2 0, E3 0, E4 0}
LIN {X 509.072, Y 342.269, Z 417.787, A -110.612, B 84.801, C -94.37, E1 0, E2 0, E3 0, E4 0}
LIN {X 507.766, Y 337.463, Z 418.238, A -110.612, B 84.801, C -94.37, E1 0, E2 0, E3 0, E4 0}
LIN {X 528.693, Y 331.359, Z 418.087, A -110.612, B 84.801, C -94.37, E1 0, E2 0, E3 0, E4 0}
LIN {X 510.536, Y 331.468, Z 418.66, A -110.612, B 84.801, C -94.37, E1 0, E2 0, E3 0, E4 0}
LIN {X 506.421, Y 332.668, Z 418.689, A -110.612, B 84.801, C -94.37, E1 0, E2 0, E3 0, E4 0}
LIN {X 593.677, Y 345.72, Z 414.783, A -110.612, B 84.801, C -94.37, E1 0, E2 0, E3 0, E4 0}
LIN {X 593.607, Y 345.536, Z 412.618, A -110.612, B 84.801, C -94.37, E1 0, E2 0, E3 0, E4 0}
LIN {X 588.564, Y 328.995, Z 414.188, A -110.612, B 84.801, C -94.37, E1 0, E2 0, E3 0, E4 0}
LIN {X 506.6, Y 331.605, Z 416.591, A -110.612, B 84.801, C -94.37, E1 0, E2 0, E3 0, E4 0}
LIN {X 505.237, Y 331.765, Z 416.621, A -110.612, B 84.801, C -94.37, E1 0, E2 0, E3 0, E4 0}
LIN {X 515.043, Y 369.337, Z 413.107, A -110.612, B 84.801, C -94.37, E1 0, E2 0, E3 0, E4 0}
LIN {X 517.381, Y 372.639, Z 412.751, A -110.612, B 84.801, C -94.37, E1 0, E2 0, E3 0, E4 0}
LIN {X 530.242, Y 370.375, Z 412.532, A -110.612, B 84.801, C -94.37, E1 0, E2 0, E3 0, E4 0}
LIN {X 531.882, Y 370.488, Z 412.47, A -110.612, B 84.801, C -94.37, E1 0, E2 0, E3 0, E4 0}
LIN {X 543.586, Y 367.702, Z 412.332, A -110.612, B 84.801, C -94.37, E1 0, E2 0, E3 0, E4 0}
LIN {X 545.643, Y 367.891, Z 412.25, A -110.612, B 84.801, C -94.37, E1 0, E2 0, E3 0, E4 0}
LIN {X 548.755, Y 367.186, Z 412.211, A -110.612, B 84.801, C -94.37, E1 0, E2 0, E3 0, E4 0}
LIN {X 549.785, Y 365.959, Z 412.282, A -110.612, B 84.801, C -94.37, E1 0, E2 0, E3 0, E4 0}
LIN {X 552.565, Y 365.277, Z 412.251, A -110.612, B 84.801, C -94.37, E1 0, E2 0, E3 0, E4 0}
LIN {X 555.211, Y 365.385, Z 412.157, A -110.612, B 84.801, C -94.37, E1 0, E2 0, E3 0, E4 0}
LIN {X 556.194, Y 365.131, Z 412.147, A -110.612, B 84.801, C -94.37, E1 0, E2 0, E3 0, E4 0}
LIN {X 556.972, Y 365.149, Z 412.121, A -110.612, B 84.801, C -94.37, E1 0, E2 0, E3 0, E4 0}
LIN {X 557.528, Y 365.488, Z 412.074, A -110.612, B 84.801, C -94.37, E1 0, E2 0, E3 0, E4 0}
LIN {X 557.721, Y 365.756, Z 412.045, A -110.612, B 84.801, C -94.37, E1 0, E2 0, E3 0, E4 0}
LIN {X 561.508, Y 364.948, Z 411.993, A -110.612, B 84.801, C -94.37, E1 0, E2 0, E3 0, E4 0}
LIN {X 562.447, Y 364.117, Z 412.034, A -110.612, B 84.801, C -94.37, E1 0, E2 0, E3 0, E4 0}
LIN {X 562.654, Y 364.019, Z 412.035, A -110.612, B 84.801, C -94.37, E1 0, E2 0, E3 0, E4 0}
LIN {X 567.794, Y 363.479, Z 411.917, A -110.612, B 84.801, C -94.37, E1 0, E2 0, E3 0, E4 0}
LIN {X 575.581, Y 361.362, Z 411.848, A -110.612, B 84.801, C -94.37, E1 0, E2 0, E3 0, E4 0}
LIN {X 577.105, Y 360.614, Z 411.862, A -110.612, B 84.801, C -94.37, E1 0, E2 0, E3 0, E4 0}
LIN {X 578.245, Y 360.715, Z 411.817, A -110.612, B 84.801, C -94.37, E1 0, E2 0, E3 0, E4 0}
LIN {X 578.517, Y 360.933, Z 411.79, A -110.612, B 84.801, C -94.37, E1 0, E2 0, E3 0, E4 0}
LIN {X 580.895, Y 360.985, Z 411.71, A -110.612, B 84.801, C -94.37, E1 0, E2 0, E3 0, E4 0}
LIN {X 586.224, Y 359.718, Z 411.647, A -110.612, B 84.801, C -94.37, E1 0, E2 0, E3 0, E4 0}
LIN {X 587.215, Y 359.054, Z 411.671, A -110.612, B 84.801, C -94.37, E1 0, E2 0, E3 0, E4 0}
LIN {X 588.479, Y 358.921, Z 411.642, A -110.612, B 84.801, C -94.37, E1 0, E2 0, E3 0, E4 0}
LIN {X 588.538, Y 358.937, Z 411.639, A -110.612, B 84.801, C -94.37, E1 0, E2 0, E3 0, E4 0}
LIN {X 593.616, Y 358.381, Z 411.524, A -110.612, B 84.801, C -94.37, E1 0, E2 0, E3 0, E4 0}
LIN {X 595.171, Y 358.68, Z 411.448, A -110.612, B 84.801, C -94.37, E1 0, E2 0, E3 0, E4 0}
LIN {X 596.506, Y 357.8, Z 411.48, A -110.612, B 84.801, C -94.37, E1 0, E2 0, E3 0, E4 0}
LIN {X 596.834, Y 356.897, Z 411.547, A -110.612, B 84.801, C -94.37, E1 0, E2 0, E3 0, E4 0}
LIN {X 596.76, Y 355.875, Z 411.636, A -110.612, B 84.801, C -94.37, E1 0, E2 0, E3 0, E4 0}
LIN {X 593.607, Y 345.536, Z 412.618, A -110.612, B 84.801, C -94.37, E1 0, E2 0, E3 0, E4 0}
LIN {X 595.801, Y 358.265, Z 411.463, A -110.612, B 84.801, C -94.37, E1 0, E2 0, E3 0, E4 0}
LIN {X 594.691, Y 358.589, Z 411.471, A -110.612, B 84.801, C -94.37, E1 0, E2 0, E3 0, E4 0}
LIN {X 553.839, Y 365.317, Z 412.207, A -110.612, B 84.801, C -94.37, E1 0, E2 0, E3 0, E4 0}
LIN {X 595.986, Y 353.024, Z 411.904, A -110.612, B 84.801, C -94.37, E1 0, E2 0, E3 0, E4 0}
LIN {X 549.15, Y 366.684, Z 412.241, A -110.612, B 84.801, C -94.37, E1 0, E2 0, E3 0, E4 0}
LIN {X 545.197, Y 367.837, Z 412.269, A -110.612, B 84.801, C -94.37, E1 0, E2 0, E3 0, E4 0}
LIN {X 516.002, Y 371.165, Z 412.921, A -110.612, B 84.801, C -94.37, E1 0, E2 0, E3 0, E4 0}
LIN {X 594.856, Y 348.167, Z 412.354, A -110.612, B 84.801, C -94.37, E1 0, E2 0, E3 0, E4 0}
LIN {X 592.931, Y 343.541, Z 412.81, A -110.612, B 84.801, C -94.37, E1 0, E2 0, E3 0, E4 0}
LIN {X 514.622, Y 366.381, Z 413.373, A -110.612, B 84.801, C -94.37, E1 0, E2 0, E3 0, E4 0}
LIN {X 513.49, Y 361.524, Z 413.822, A -110.612, B 84.801, C -94.37, E1 0, E2 0, E3 0, E4 0}
LIN {X 591.509, Y 338.769, Z 413.261, A -110.612, B 84.801, C -94.37, E1 0, E2 0, E3 0, E4 0}
LIN {X 590.259, Y 333.946, Z 413.712, A -110.612, B 84.801, C -94.37, E1 0, E2 0, E3 0, E4 0}
LIN {X 512.104, Y 356.741, Z 414.274, A -110.612, B 84.801, C -94.37, E1 0, E2 0, E3 0, E4 0}
LIN {X 510.988, Y 351.88, Z 414.724, A -110.612, B 84.801, C -94.37, E1 0, E2 0, E3 0, E4 0}
LIN {X 588.624, Y 329.236, Z 414.166, A -110.612, B 84.801, C -94.37, E1 0, E2 0, E3 0, E4 0}
LIN {X 567.266, Y 330.279, Z 414.761, A -110.612, B 84.801, C -94.37, E1 0, E2 0, E3 0, E4 0}
LIN {X 567.245, Y 330.285, Z 414.761, A -110.612, B 84.801, C -94.37, E1 0, E2 0, E3 0, E4 0}
LIN {X 509.789, Y 347.042, Z 415.174, A -110.612, B 84.801, C -94.37, E1 0, E2 0, E3 0, E4 0}
LIN {X 508.271, Y 342.298, Z 415.627, A -110.612, B 84.801, C -94.37, E1 0, E2 0, E3 0, E4 0}
LIN {X 546.753, Y 331.074, Z 415.35, A -110.612, B 84.801, C -94.37, E1 0, E2 0, E3 0, E4 0}
LIN {X 528.68, Y 331.158, Z 415.922, A -110.612, B 84.801, C -94.37, E1 0, E2 0, E3 0, E4 0}
LIN {X 507.076, Y 337.459, Z 416.077, A -110.612, B 84.801, C -94.37, E1 0, E2 0, E3 0, E4 0}
LIN {X 505.576, Y 332.71, Z 416.53, A -110.612, B 84.801, C -94.37, E1 0, E2 0, E3 0, E4 0}
LIN {X 510.576, Y 331.251, Z 416.494, A -110.612, B 84.801, C -94.37, E1 0, E2 0, E3 0, E4 0}
LIN {X 594.741, Y 345.204, Z 412.61, A -110.612, B 84.801, C -94.37, E1 0, E2 0, E3 0, E4 0}
LIN {X 594.671, Y 345.02, Z 410.445, A -110.612, B 84.801, C -94.37, E1 0, E2 0, E3 0, E4 0}
LIN {X 589.928, Y 328.795, Z 411.979, A -110.612, B 84.801, C -94.37, E1 0, E2 0, E3 0, E4 0}
LIN {X 509.164, Y 331.168, Z 414.363, A -110.612, B 84.801, C -94.37, E1 0, E2 0, E3 0, E4 0}
LIN {X 504.673, Y 331.627, Z 414.468, A -110.612, B 84.801, C -94.37, E1 0, E2 0, E3 0, E4 0}
LIN {X 515.354, Y 371.285, Z 410.749, A -110.612, B 84.801, C -94.37, E1 0, E2 0, E3 0, E4 0}
LIN {X 516.557, Y 372.528, Z 410.604, A -110.612, B 84.801, C -94.37, E1 0, E2 0, E3 0, E4 0}
LIN {X 517.034, Y 372.541, Z 410.588, A -110.612, B 84.801, C -94.37, E1 0, E2 0, E3 0, E4 0}
LIN {X 518.742, Y 372.032, Z 410.577, A -110.612, B 84.801, C -94.37, E1 0, E2 0, E3 0, E4 0}
LIN {X 519.145, Y 372.084, Z 410.559, A -110.612, B 84.801, C -94.37, E1 0, E2 0, E3 0, E4 0}
LIN {X 520.343, Y 372.615, Z 410.476, A -110.612, B 84.801, C -94.37, E1 0, E2 0, E3 0, E4 0}
LIN {X 544.517, Y 367.893, Z 410.104, A -110.612, B 84.801, C -94.37, E1 0, E2 0, E3 0, E4 0}
LIN {X 544.694, Y 367.754, Z 410.11, A -110.612, B 84.801, C -94.37, E1 0, E2 0, E3 0, E4 0}
LIN {X 546.396, Y 367.701, Z 410.06, A -110.612, B 84.801, C -94.37, E1 0, E2 0, E3 0, E4 0}
LIN {X 551.445, Y 366.479, Z 410.002, A -110.612, B 84.801, C -94.37, E1 0, E2 0, E3 0, E4 0}
LIN {X 551.725, Y 366.331, Z 410.006, A -110.612, B 84.801, C -94.37, E1 0, E2 0, E3 0, E4 0}
LIN {X 554.353, Y 366.047, Z 409.946, A -110.612, B 84.801, C -94.37, E1 0, E2 0, E3 0, E4 0}
LIN {X 554.562, Y 366.104, Z 409.934, A -110.612, B 84.801, C -94.37, E1 0, E2 0, E3 0, E4 0}
LIN {X 560.267, Y 365.427, Z 409.809, A -110.612, B 84.801, C -94.37, E1 0, E2 0, E3 0, E4 0}
LIN {X 562.537, Y 364.221, Z 409.839, A -110.612, B 84.801, C -94.37, E1 0, E2 0, E3 0, E4 0}
LIN {X 564.622, Y 363.667, Z 409.819, A -110.612, B 84.801, C -94.37, E1 0, E2 0, E3 0, E4 0}
LIN {X 564.753, Y 363.741, Z 409.809, A -110.612, B 84.801, C -94.37, E1 0, E2 0, E3 0, E4 0}
LIN {X 577.155, Y 361.335, Z 409.617, A -110.612, B 84.801, C -94.37, E1 0, E2 0, E3 0, E4 0}
LIN {X 577.565, Y 361.523, Z 409.587, A -110.612, B 84.801, C -94.37, E1 0, E2 0, E3 0, E4 0}
LIN {X 578.306, Y 361.56, Z 409.561, A -110.612, B 84.801, C -94.37, E1 0, E2 0, E3 0, E4 0}
LIN {X 584.696, Y 359.716, Z 409.513, A -110.612, B 84.801, C -94.37, E1 0, E2 0, E3 0, E4 0}
LIN {X 597.151, Y 357.772, Z 409.28, A -110.612, B 84.801, C -94.37, E1 0, E2 0, E3 0, E4 0}
LIN {X 597.696, Y 357.455, Z 409.289, A -110.612, B 84.801, C -94.37, E1 0, E2 0, E3 0, E4 0}
LIN {X 598.035, Y 356.547, Z 409.356, A -110.612, B 84.801, C -94.37, E1 0, E2 0, E3 0, E4 0}
LIN {X 598.036, Y 356.529, Z 409.357, A -110.612, B 84.801, C -94.37, E1 0, E2 0, E3 0, E4 0}
LIN {X 594.671, Y 345.02, Z 410.445, A -110.612, B 84.801, C -94.37, E1 0, E2 0, E3 0, E4 0}
LIN {X 597.513, Y 357.561, Z 409.286, A -110.612, B 84.801, C -94.37, E1 0, E2 0, E3 0, E4 0}
LIN {X 596.245, Y 357.931, Z 409.295, A -110.612, B 84.801, C -94.37, E1 0, E2 0, E3 0, E4 0}
LIN {X 544.85, Y 367.734, Z 410.107, A -110.612, B 84.801, C -94.37, E1 0, E2 0, E3 0, E4 0}
LIN {X 597.237, Y 352.455, Z 409.73, A -110.612, B 84.801, C -94.37, E1 0, E2 0, E3 0, E4 0}
LIN {X 544.643, Y 367.794, Z 410.108, A -110.612, B 84.801, C -94.37, E1 0, E2 0, E3 0, E4 0}
LIN {X 543.702, Y 368.069, Z 410.115, A -110.612, B 84.801, C -94.37, E1 0, E2 0, E3 0, E4 0}
LIN {X 515.301, Y 371.165, Z 410.761, A -110.612, B 84.801, C -94.37, E1 0, E2 0, E3 0, E4 0}
LIN {X 595.916, Y 347.653, Z 410.181, A -110.612, B 84.801, C -94.37, E1 0, E2 0, E3 0, E4 0}
LIN {X 594.161, Y 342.978, Z 410.635, A -110.612, B 84.801, C -94.37, E1 0, E2 0, E3 0, E4 0}
LIN {X 513.516, Y 366.499, Z 411.215, A -110.612, B 84.801, C -94.37, E1 0, E2 0, E3 0, E4 0}
LIN {X 512.298, Y 361.667, Z 411.666, A -110.612, B 84.801, C -94.37, E1 0, E2 0, E3 0, E4 0}
LIN {X 592.832, Y 338.178, Z 411.087, A -110.612, B 84.801, C -94.37, E1 0, E2 0, E3 0, E4 0}
LIN {X 591.46, Y 333.392, Z 411.538, A -110.612, B 84.801, C -94.37, E1 0, E2 0, E3 0, E4 0}
LIN {X 511.321, Y 356.765, Z 412.114, A -110.612, B 84.801, C -94.37, E1 0, E2 0, E3 0, E4 0}
LIN {X 510.194, Y 351.906, Z 412.564, A -110.612, B 84.801, C -94.37, E1 0, E2 0, E3 0, E4 0}
LIN {X 589.426, Y 328.798, Z 411.995, A -110.612, B 84.801, C -94.37, E1 0, E2 0, E3 0, E4 0}
LIN {X 567.25, Y 330.078, Z 412.596, A -110.612, B 84.801, C -94.37, E1 0, E2 0, E3 0, E4 0}
LIN {X 509.203, Y 347.009, Z 413.013, A -110.612, B 84.801, C -94.37, E1 0, E2 0, E3 0, E4 0}
LIN {X 507.762, Y 342.242, Z 413.465, A -110.612, B 84.801, C -94.37, E1 0, E2 0, E3 0, E4 0}
LIN {X 546.713, Y 330.881, Z 413.185, A -110.612, B 84.801, C -94.37, E1 0, E2 0, E3 0, E4 0}
LIN {X 528.626, Y 330.97, Z 413.757, A -110.612, B 84.801, C -94.37, E1 0, E2 0, E3 0, E4 0}
LIN {X 506.343, Y 337.469, Z 413.917, A -110.612, B 84.801, C -94.37, E1 0, E2 0, E3 0, E4 0}
LIN {X 504.978, Y 332.68, Z 414.369, A -110.612, B 84.801, C -94.37, E1 0, E2 0, E3 0, E4 0}
LIN {X 510.559, Y 331.052, Z 414.328, A -110.612, B 84.801, C -94.37, E1 0, E2 0, E3 0, E4 0}
LIN {X 595.711, Y 344.735, Z 410.436, A -110.612, B 84.801, C -94.37, E1 0, E2 0, E3 0, E4 0}
LIN {X 595.642, Y 344.551, Z 408.271, A -110.612, B 84.801, C -94.37, E1 0, E2 0, E3 0, E4 0}
LIN {X 591.291, Y 328.582, Z 409.77, A -110.612, B 84.801, C -94.37, E1 0, E2 0, E3 0, E4 0}
LIN {X 506.402, Y 331.208, Z 412.265, A -110.612, B 84.801, C -94.37, E1 0, E2 0, E3 0, E4 0}
LIN {X 504.059, Y 331.507, Z 412.315, A -110.612, B 84.801, C -94.37, E1 0, E2 0, E3 0, E4 0}
LIN {X 514.786, Y 371.138, Z 408.596, A -110.612, B 84.801, C -94.37, E1 0, E2 0, E3 0, E4 0}
LIN {X 515.485, Y 372.123, Z 408.49, A -110.612, B 84.801, C -94.37, E1 0, E2 0, E3 0, E4 0}
LIN {X 516.392, Y 372.739, Z 408.409, A -110.612, B 84.801, C -94.37, E1 0, E2 0, E3 0, E4 0}
LIN {X 518.28, Y 372.869, Z 408.337, A -110.612, B 84.801, C -94.37, E1 0, E2 0, E3 0, E4 0}
LIN {X 522.371, Y 372.023, Z 408.278, A -110.612, B 84.801, C -94.37, E1 0, E2 0, E3 0, E4 0}
LIN {X 522.419, Y 372.035, Z 408.276, A -110.612, B 84.801, C -94.37, E1 0, E2 0, E3 0, E4 0}
LIN {X 532.773, Y 369.805, Z 408.134, A -110.612, B 84.801, C -94.37, E1 0, E2 0, E3 0, E4 0}
LIN {X 532.899, Y 369.828, Z 408.128, A -110.612, B 84.801, C -94.37, E1 0, E2 0, E3 0, E4 0}
LIN {X 539.166, Y 368.476, Z 408.042, A -110.612, B 84.801, C -94.37, E1 0, E2 0, E3 0, E4 0}
LIN {X 540.061, Y 368.722, Z 407.993, A -110.612, B 84.801, C -94.37, E1 0, E2 0, E3 0, E4 0}
LIN {X 549.924, Y 366.614, Z 407.856, A -110.612, B 84.801, C -94.37, E1 0, E2 0, E3 0, E4 0}
LIN {X 550.805, Y 365.898, Z 407.889, A -110.612, B 84.801, C -94.37, E1 0, E2 0, E3 0, E4 0}
LIN {X 552.919, Y 365.397, Z 407.864, A -110.612, B 84.801, C -94.37, E1 0, E2 0, E3 0, E4 0}
LIN {X 553.152, Y 365.527, Z 407.846, A -110.612, B 84.801, C -94.37, E1 0, E2 0, E3 0, E4 0}
LIN {X 554.596, Y 365.508, Z 407.801, A -110.612, B 84.801, C -94.37, E1 0, E2 0, E3 0, E4 0}
LIN {X 555.163, Y 365.32, Z 407.799, A -110.612, B 84.801, C -94.37, E1 0, E2 0, E3 0, E4 0}
LIN {X 560.135, Y 365.327, Z 407.639, A -110.612, B 84.801, C -94.37, E1 0, E2 0, E3 0, E4 0}
LIN {X 560.767, Y 364.952, Z 407.651, A -110.612, B 84.801, C -94.37, E1 0, E2 0, E3 0, E4 0}
LIN {X 561.601, Y 363.796, Z 407.722, A -110.612, B 84.801, C -94.37, E1 0, E2 0, E3 0, E4 0}
LIN {X 561.696, Y 363.733, Z 407.725, A -110.612, B 84.801, C -94.37, E1 0, E2 0, E3 0, E4 0}
LIN {X 563.071, Y 363.609, Z 407.691, A -110.612, B 84.801, C -94.37, E1 0, E2 0, E3 0, E4 0}
LIN {X 564.986, Y 362.679, Z 407.709, A -110.612, B 84.801, C -94.37, E1 0, E2 0, E3 0, E4 0}
LIN {X 566.277, Y 362.756, Z 407.661, A -110.612, B 84.801, C -94.37, E1 0, E2 0, E3 0, E4 0}
LIN {X 566.515, Y 363.086, Z 407.625, A -110.612, B 84.801, C -94.37, E1 0, E2 0, E3 0, E4 0}
LIN {X 568.255, Y 362.884, Z 407.587, A -110.612, B 84.801, C -94.37, E1 0, E2 0, E3 0, E4 0}
LIN {X 570.014, Y 363.327, Z 407.493, A -110.612, B 84.801, C -94.37, E1 0, E2 0, E3 0, E4 0}
LIN {X 572.584, Y 362.827, Z 407.453, A -110.612, B 84.801, C -94.37, E1 0, E2 0, E3 0, E4 0}
LIN {X 573.073, Y 362.544, Z 407.462, A -110.612, B 84.801, C -94.37, E1 0, E2 0, E3 0, E4 0}
LIN {X 582.665, Y 360.502, Z 407.328, A -110.612, B 84.801, C -94.37, E1 0, E2 0, E3 0, E4 0}
LIN {X 583.707, Y 360.424, Z 407.301, A -110.612, B 84.801, C -94.37, E1 0, E2 0, E3 0, E4 0}
LIN {X 583.769, Y 360.447, Z 407.297, A -110.612, B 84.801, C -94.37, E1 0, E2 0, E3 0, E4 0}
LIN {X 597.892, Y 357.824, Z 407.068, A -110.612, B 84.801, C -94.37, E1 0, E2 0, E3 0, E4 0}
LIN {X 598.852, Y 356.88, Z 407.118, A -110.612, B 84.801, C -94.37, E1 0, E2 0, E3 0, E4 0}
LIN {X 598.936, Y 356.638, Z 407.136, A -110.612, B 84.801, C -94.37, E1 0, E2 0, E3 0, E4 0}
LIN {X 595.642, Y 344.551, Z 408.271, A -110.612, B 84.801, C -94.37, E1 0, E2 0, E3 0, E4 0}
LIN {X 593.062, Y 358.655, Z 407.152, A -110.612, B 84.801, C -94.37, E1 0, E2 0, E3 0, E4 0}
LIN {X 598.744, Y 356.998, Z 407.111, A -110.612, B 84.801, C -94.37, E1 0, E2 0, E3 0, E4 0}
LIN {X 598.302, Y 351.939, Z 407.556, A -110.612, B 84.801, C -94.37, E1 0, E2 0, E3 0, E4 0}
LIN {X 543.828, Y 367.827, Z 407.948, A -110.612, B 84.801, C -94.37, E1 0, E2 0, E3 0, E4 0}
LIN {X 514.778, Y 371.113, Z 408.599, A -110.612, B 84.801, C -94.37, E1 0, E2 0, E3 0, E4 0}
LIN {X 596.757, Y 347.203, Z 408.009, A -110.612, B 84.801, C -94.37, E1 0, E2 0, E3 0, E4 0}
LIN {X 595.319, Y 342.436, Z 408.461, A -110.612, B 84.801, C -94.37, E1 0, E2 0, E3 0, E4 0}
LIN {X 512.939, Y 366.463, Z 409.054, A -110.612, B 84.801, C -94.37, E1 0, E2 0, E3 0, E4 0}
LIN {X 511.685, Y 361.641, Z 409.505, A -110.612, B 84.801, C -94.37, E1 0, E2 0, E3 0, E4 0}
LIN {X 594.1, Y 337.604, Z 408.912, A -110.612, B 84.801, C -94.37, E1 0, E2 0, E3 0, E4 0}
LIN {X 592.623, Y 332.848, Z 409.364, A -110.612, B 84.801, C -94.37, E1 0, E2 0, E3 0, E4 0}
LIN {X 510.581, Y 356.776, Z 409.954, A -110.612, B 84.801, C -94.37, E1 0, E2 0, E3 0, E4 0}
LIN {X 509.482, Y 351.91, Z 410.404, A -110.612, B 84.801, C -94.37, E1 0, E2 0, E3 0, E4 0}
LIN {X 589.429, Y 328.592, Z 409.829, A -110.612, B 84.801, C -94.37, E1 0, E2 0, E3 0, E4 0}
LIN {X 567.291, Y 329.862, Z 410.43, A -110.612, B 84.801, C -94.37, E1 0, E2 0, E3 0, E4 0}
LIN {X 508.549, Y 346.995, Z 410.852, A -110.612, B 84.801, C -94.37, E1 0, E2 0, E3 0, E4 0}
LIN {X 507.22, Y 342.195, Z 411.304, A -110.612, B 84.801, C -94.37, E1 0, E2 0, E3 0, E4 0}
LIN {X 546.72, Y 330.675, Z 411.019, A -110.612, B 84.801, C -94.37, E1 0, E2 0, E3 0, E4 0}
LIN {X 528.612, Y 330.769, Z 411.591, A -110.612, B 84.801, C -94.37, E1 0, E2 0, E3 0, E4 0}
LIN {X 505.868, Y 337.402, Z 411.755, A -110.612, B 84.801, C -94.37, E1 0, E2 0, E3 0, E4 0}
LIN {X 504.405, Y 332.642, Z 412.207, A -110.612, B 84.801, C -94.37, E1 0, E2 0, E3 0, E4 0}
LIN {X 510.597, Y 330.836, Z 412.163, A -110.612, B 84.801, C -94.37, E1 0, E2 0, E3 0, E4 0}
LIN {X 596.566, Y 344.31, Z 408.262, A -110.612, B 84.801, C -94.37, E1 0, E2 0, E3 0, E4 0}
LIN {X 596.497, Y 344.126, Z 406.097, A -110.612, B 84.801, C -94.37, E1 0, E2 0, E3 0, E4 0}
LIN {X 599.62, Y 356.18, Z 404.97, A -110.612, B 84.801, C -94.37, E1 0, E2 0, E3 0, E4 0}
LIN {X 599.079, Y 356.977, Z 404.92, A -110.612, B 84.801, C -94.37, E1 0, E2 0, E3 0, E4 0}
LIN {X 597.005, Y 358.062, Z 404.894, A -110.612, B 84.801, C -94.37, E1 0, E2 0, E3 0, E4 0}
LIN {X 564.726, Y 364.213, Z 405.404, A -110.612, B 84.801, C -94.37, E1 0, E2 0, E3 0, E4 0}
LIN {X 563.258, Y 363.7, Z 405.494, A -110.612, B 84.801, C -94.37, E1 0, E2 0, E3 0, E4 0}
LIN {X 553.573, Y 366.089, Z 405.601, A -110.612, B 84.801, C -94.37, E1 0, E2 0, E3 0, E4 0}
LIN {X 551.851, Y 365.778, Z 405.683, A -110.612, B 84.801, C -94.37, E1 0, E2 0, E3 0, E4 0}
LIN {X 540.217, Y 368.825, Z 405.796, A -110.612, B 84.801, C -94.37, E1 0, E2 0, E3 0, E4 0}
LIN {X 539.905, Y 368.675, Z 405.819, A -110.612, B 84.801, C -94.37, E1 0, E2 0, E3 0, E4 0}
LIN {X 538.498, Y 369.079, Z 405.829, A -110.612, B 84.801, C -94.37, E1 0, E2 0, E3 0, E4 0}
LIN {X 532.805, Y 369.33, Z 405.99, A -110.612, B 84.801, C -94.37, E1 0, E2 0, E3 0, E4 0}
LIN {X 532.63, Y 369.265, Z 406.002, A -110.612, B 84.801, C -94.37, E1 0, E2 0, E3 0, E4 0}
LIN {X 530.985, Y 369.272, Z 406.054, A -110.612, B 84.801, C -94.37, E1 0, E2 0, E3 0, E4 0}
LIN {X 528.96, Y 370.529, Z 406.011, A -110.612, B 84.801, C -94.37, E1 0, E2 0, E3 0, E4 0}
LIN {X 521.042, Y 372.243, Z 406.119, A -110.612, B 84.801, C -94.37, E1 0, E2 0, E3 0, E4 0}
LIN {X 520.774, Y 372.176, Z 406.133, A -110.612, B 84.801, C -94.37, E1 0, E2 0, E3 0, E4 0}
LIN {X 518.626, Y 372.722, Z 406.156, A -110.612, B 84.801, C -94.37, E1 0, E2 0, E3 0, E4 0}
LIN {X 518.561, Y 372.689, Z 406.161, A -110.612, B 84.801, C -94.37, E1 0, E2 0, E3 0, E4 0}
LIN {X 518.47, Y 372.787, Z 406.155, A -110.612, B 84.801, C -94.37, E1 0, E2 0, E3 0, E4 0}
LIN {X 516.086, Y 372.797, Z 406.231, A -110.612, B 84.801, C -94.37, E1 0, E2 0, E3 0, E4 0}
LIN {X 515.311, Y 372.287, Z 406.299, A -110.612, B 84.801, C -94.37, E1 0, E2 0, E3 0, E4 0}
LIN {X 514.414, Y 371.13, Z 406.426, A -110.612, B 84.801, C -94.37, E1 0, E2 0, E3 0, E4 0}
LIN {X 503.814, Y 331.74, Z 410.12, A -110.612, B 84.801, C -94.37, E1 0, E2 0, E3 0, E4 0}
LIN {X 503.748, Y 331.355, Z 410.155, A -110.612, B 84.801, C -94.37, E1 0, E2 0, E3 0, E4 0}
LIN {X 504.382, Y 331.244, Z 410.144, A -110.612, B 84.801, C -94.37, E1 0, E2 0, E3 0, E4 0}
LIN {X 592.414, Y 328.37, Z 407.569, A -110.612, B 84.801, C -94.37, E1 0, E2 0, E3 0, E4 0}
LIN {X 596.497, Y 344.126, Z 406.097, A -110.612, B 84.801, C -94.37, E1 0, E2 0, E3 0, E4 0}
LIN {X 589.706, Y 359.429, Z 405.011, A -110.612, B 84.801, C -94.37, E1 0, E2 0, E3 0, E4 0}
LIN {X 599.364, Y 356.612, Z 404.942, A -110.612, B 84.801, C -94.37, E1 0, E2 0, E3 0, E4 0}
LIN {X 599.159, Y 351.485, Z 405.385, A -110.612, B 84.801, C -94.37, E1 0, E2 0, E3 0, E4 0}
LIN {X 540.024, Y 368.732, Z 405.81, A -110.612, B 84.801, C -94.37, E1 0, E2 0, E3 0, E4 0}
LIN {X 514.381, Y 371.024, Z 406.436, A -110.612, B 84.801, C -94.37, E1 0, E2 0, E3 0, E4 0}
LIN {X 597.957, Y 346.649, Z 405.835, A -110.612, B 84.801, C -94.37, E1 0, E2 0, E3 0, E4 0}
LIN {X 596.463, Y 341.897, Z 406.288, A -110.612, B 84.801, C -94.37, E1 0, E2 0, E3 0, E4 0}
LIN {X 512.653, Y 366.341, Z 406.89, A -110.612, B 84.801, C -94.37, E1 0, E2 0, E3 0, E4 0}
LIN {X 511.122, Y 361.601, Z 407.343, A -110.612, B 84.801, C -94.37, E1 0, E2 0, E3 0, E4 0}
LIN {X 595.192, Y 337.081, Z 406.739, A -110.612, B 84.801, C -94.37, E1 0, E2 0, E3 0, E4 0}
LIN {X 593.592, Y 332.36, Z 407.192, A -110.612, B 84.801, C -94.37, E1 0, E2 0, E3 0, E4 0}
LIN {X 510.103, Y 356.711, Z 407.792, A -110.612, B 84.801, C -94.37, E1 0, E2 0, E3 0, E4 0}
LIN {X 509.017, Y 351.841, Z 408.242, A -110.612, B 84.801, C -94.37, E1 0, E2 0, E3 0, E4 0}
LIN {X 589.381, Y 328.402, Z 407.664, A -110.612, B 84.801, C -94.37, E1 0, E2 0, E3 0, E4 0}
LIN {X 567.262, Y 329.666, Z 408.264, A -110.612, B 84.801, C -94.37, E1 0, E2 0, E3 0, E4 0}
LIN {X 508.08, Y 346.927, Z 408.69, A -110.612, B 84.801, C -94.37, E1 0, E2 0, E3 0, E4 0}
LIN {X 506.821, Y 342.107, Z 409.141, A -110.612, B 84.801, C -94.37, E1 0, E2 0, E3 0, E4 0}
LIN {X 546.673, Y 330.484, Z 408.854, A -110.612, B 84.801, C -94.37, E1 0, E2 0, E3 0, E4 0}
LIN {X 528.555, Y 330.581, Z 409.426, A -110.612, B 84.801, C -94.37, E1 0, E2 0, E3 0, E4 0}
LIN {X 505.52, Y 337.299, Z 409.592, A -110.612, B 84.801, C -94.37, E1 0, E2 0, E3 0, E4 0}
LIN {X 504.056, Y 332.539, Z 410.044, A -110.612, B 84.801, C -94.37, E1 0, E2 0, E3 0, E4 0}
LIN {X 510.566, Y 330.641, Z 409.997, A -110.612, B 84.801, C -94.37, E1 0, E2 0, E3 0, E4 0}
LIN {X 597.171, Y 343.959, Z 406.09, A -110.612, B 84.801, C -94.37, E1 0, E2 0, E3 0, E4 0}
LIN {X 597.101, Y 343.774, Z 403.925, A -110.612, B 84.801, C -94.37, E1 0, E2 0, E3 0, E4 0}
LIN {X 593.233, Y 328.154, Z 405.379, A -110.612, B 84.801, C -94.37, E1 0, E2 0, E3 0, E4 0}
LIN {X 593.206, Y 328.145, Z 405.38, A -110.612, B 84.801, C -94.37, E1 0, E2 0, E3 0, E4 0}
LIN {X 506.215, Y 330.821, Z 407.939, A -110.612, B 84.801, C -94.37, E1 0, E2 0, E3 0, E4 0}
LIN {X 503.796, Y 331.133, Z 407.989, A -110.612, B 84.801, C -94.37, E1 0, E2 0, E3 0, E4 0}
LIN {X 513.633, Y 369.86, Z 404.377, A -110.612, B 84.801, C -94.37, E1 0, E2 0, E3 0, E4 0}
LIN {X 515.332, Y 372.376, Z 404.108, A -110.612, B 84.801, C -94.37, E1 0, E2 0, E3 0, E4 0}
LIN {X 516.255, Y 372.942, Z 404.03, A -110.612, B 84.801, C -94.37, E1 0, E2 0, E3 0, E4 0}
LIN {X 523.932, Y 371.671, Z 403.892, A -110.612, B 84.801, C -94.37, E1 0, E2 0, E3 0, E4 0}
LIN {X 525.317, Y 369.987, Z 403.991, A -110.612, B 84.801, C -94.37, E1 0, E2 0, E3 0, E4 0}
LIN {X 527.872, Y 369.291, Z 403.969, A -110.612, B 84.801, C -94.37, E1 0, E2 0, E3 0, E4 0}
LIN {X 528.975, Y 369.241, Z 403.938, A -110.612, B 84.801, C -94.37, E1 0, E2 0, E3 0, E4 0}
LIN {X 530.235, Y 368.592, Z 403.953, A -110.612, B 84.801, C -94.37, E1 0, E2 0, E3 0, E4 0}
LIN {X 530.597, Y 368.824, Z 403.921, A -110.612, B 84.801, C -94.37, E1 0, E2 0, E3 0, E4 0}
LIN {X 531.057, Y 369.349, Z 403.862, A -110.612, B 84.801, C -94.37, E1 0, E2 0, E3 0, E4 0}
LIN {X 533.947, Y 369.468, Z 403.759, A -110.612, B 84.801, C -94.37, E1 0, E2 0, E3 0, E4 0}
LIN {X 538.36, Y 368.539, Z 403.697, A -110.612, B 84.801, C -94.37, E1 0, E2 0, E3 0, E4 0}
LIN {X 540.011, Y 368.7, Z 403.63, A -110.612, B 84.801, C -94.37, E1 0, E2 0, E3 0, E4 0}
LIN {X 544.394, Y 367.895, Z 403.559, A -110.612, B 84.801, C -94.37, E1 0, E2 0, E3 0, E4 0}
LIN {X 544.813, Y 367.641, Z 403.567, A -110.612, B 84.801, C -94.37, E1 0, E2 0, E3 0, E4 0}
LIN {X 546.413, Y 367.46, Z 403.531, A -110.612, B 84.801, C -94.37, E1 0, E2 0, E3 0, E4 0}
LIN {X 548.166, Y 366.809, Z 403.53, A -110.612, B 84.801, C -94.37, E1 0, E2 0, E3 0, E4 0}
LIN {X 549.889, Y 366.761, Z 403.479, A -110.612, B 84.801, C -94.37, E1 0, E2 0, E3 0, E4 0}
LIN {X 551.327, Y 366.165, Z 403.484, A -110.612, B 84.801, C -94.37, E1 0, E2 0, E3 0, E4 0}
LIN {X 555.145, Y 366.232, Z 403.356, A -110.612, B 84.801, C -94.37, E1 0, E2 0, E3 0, E4 0}
LIN {X 558.13, Y 365.206, Z 403.348, A -110.612, B 84.801, C -94.37, E1 0, E2 0, E3 0, E4 0}
LIN {X 559.091, Y 363.841, Z 403.433, A -110.612, B 84.801, C -94.37, E1 0, E2 0, E3 0, E4 0}
LIN {X 561.347, Y 363.661, Z 403.376, A -110.612, B 84.801, C -94.37, E1 0, E2 0, E3 0, E4 0}
LIN {X 562.982, Y 364.281, Z 403.271, A -110.612, B 84.801, C -94.37, E1 0, E2 0, E3 0, E4 0}
LIN {X 571.589, Y 362.455, Z 403.151, A -110.612, B 84.801, C -94.37, E1 0, E2 0, E3 0, E4 0}
LIN {X 571.618, Y 362.467, Z 403.149, A -110.612, B 84.801, C -94.37, E1 0, E2 0, E3 0, E4 0}
LIN {X 573.109, Y 362.333, Z 403.113, A -110.612, B 84.801, C -94.37, E1 0, E2 0, E3 0, E4 0}
LIN {X 574.336, Y 361.791, Z 403.119, A -110.612, B 84.801, C -94.37, E1 0, E2 0, E3 0, E4 0}
LIN {X 575.757, Y 361.661, Z 403.085, A -110.612, B 84.801, C -94.37, E1 0, E2 0, E3 0, E4 0}
LIN {X 575.927, Y 361.687, Z 403.077, A -110.612, B 84.801, C -94.37, E1 0, E2 0, E3 0, E4 0}
LIN {X 596.769, Y 358.185, Z 402.708, A -110.612, B 84.801, C -94.37, E1 0, E2 0, E3 0, E4 0}
LIN {X 599.475, Y 356.537, Z 402.762, A -110.612, B 84.801, C -94.37, E1 0, E2 0, E3 0, E4 0}
LIN {X 599.631, Y 356.286, Z 402.778, A -110.612, B 84.801, C -94.37, E1 0, E2 0, E3 0, E4 0}
LIN {X 599.904, Y 355.091, Z 402.871, A -110.612, B 84.801, C -94.37, E1 0, E2 0, E3 0, E4 0}
LIN {X 597.101, Y 343.774, Z 403.925, A -110.612, B 84.801, C -94.37, E1 0, E2 0, E3 0, E4 0}
LIN {X 587.64, Y 359.827, Z 402.861, A -110.612, B 84.801, C -94.37, E1 0, E2 0, E3 0, E4 0}
LIN {X 599.598, Y 356.339, Z 402.775, A -110.612, B 84.801, C -94.37, E1 0, E2 0, E3 0, E4 0}
LIN {X 599.248, Y 351.255, Z 403.219, A -110.612, B 84.801, C -94.37, E1 0, E2 0, E3 0, E4 0}
LIN {X 539.695, Y 368.624, Z 403.647, A -110.612, B 84.801, C -94.37, E1 0, E2 0, E3 0, E4 0}
LIN {X 514.179, Y 370.879, Z 404.272, A -110.612, B 84.801, C -94.37, E1 0, E2 0, E3 0, E4 0}
LIN {X 598.141, Y 346.39, Z 403.668, A -110.612, B 84.801, C -94.37, E1 0, E2 0, E3 0, E4 0}
LIN {X 596.981, Y 341.542, Z 404.119, A -110.612, B 84.801, C -94.37, E1 0, E2 0, E3 0, E4 0}
LIN {X 512.315, Y 366.235, Z 404.727, A -110.612, B 84.801, C -94.37, E1 0, E2 0, E3 0, E4 0}
LIN {X 510.918, Y 361.456, Z 405.179, A -110.612, B 84.801, C -94.37, E1 0, E2 0, E3 0, E4 0}
LIN {X 595.625, Y 336.75, Z 404.57, A -110.612, B 84.801, C -94.37, E1 0, E2 0, E3 0, E4 0}
LIN {X 594.478, Y 331.898, Z 405.02, A -110.612, B 84.801, C -94.37, E1 0, E2 0, E3 0, E4 0}
LIN {X 509.793, Y 356.597, Z 405.629, A -110.612, B 84.801, C -94.37, E1 0, E2 0, E3 0, E4 0}
LIN {X 508.84, Y 351.688, Z 406.077, A -110.612, B 84.801, C -94.37, E1 0, E2 0, E3 0, E4 0}
LIN {X 589.357, Y 328.204, Z 405.499, A -110.612, B 84.801, C -94.37, E1 0, E2 0, E3 0, E4 0}
LIN {X 567.266, Y 329.46, Z 406.099, A -110.612, B 84.801, C -94.37, E1 0, E2 0, E3 0, E4 0}
LIN {X 507.926, Y 346.767, Z 406.526, A -110.612, B 84.801, C -94.37, E1 0, E2 0, E3 0, E4 0}
LIN {X 506.658, Y 341.95, Z 406.977, A -110.612, B 84.801, C -94.37, E1 0, E2 0, E3 0, E4 0}
LIN {X 546.652, Y 330.285, Z 406.689, A -110.612, B 84.801, C -94.37, E1 0, E2 0, E3 0, E4 0}
LIN {X 528.518, Y 330.387, Z 407.261, A -110.612, B 84.801, C -94.37, E1 0, E2 0, E3 0, E4 0}
LIN {X 505.372, Y 337.138, Z 407.428, A -110.612, B 84.801, C -94.37, E1 0, E2 0, E3 0, E4 0}
LIN {X 504.102, Y 332.321, Z 407.878, A -110.612, B 84.801, C -94.37, E1 0, E2 0, E3 0, E4 0}
LIN {X 510.568, Y 330.436, Z 407.832, A -110.612, B 84.801, C -94.37, E1 0, E2 0, E3 0, E4 0}
LIN {X 597.297, Y 343.731, Z 403.922, A -110.612, B 84.801, C -94.37, E1 0, E2 0, E3 0, E4 0}
LIN {X 597.227, Y 343.546, Z 401.757, A -110.612, B 84.801, C -94.37, E1 0, E2 0, E3 0, E4 0}
LIN {X 599.896, Y 355.543, Z 400.65, A -110.612, B 84.801, C -94.37, E1 0, E2 0, E3 0, E4 0}
LIN {X 599.16, Y 356.917, Z 400.557, A -110.612, B 84.801, C -94.37, E1 0, E2 0, E3 0, E4 0}
LIN {X 597.296, Y 357.904, Z 400.532, A -110.612, B 84.801, C -94.37, E1 0, E2 0, E3 0, E4 0}
LIN {X 583.016, Y 360.386, Z 400.778, A -110.612, B 84.801, C -94.37, E1 0, E2 0, E3 0, E4 0}
LIN {X 581.885, Y 359.983, Z 400.849, A -110.612, B 84.801, C -94.37, E1 0, E2 0, E3 0, E4 0}
LIN {X 572.725, Y 361.954, Z 400.974, A -110.612, B 84.801, C -94.37, E1 0, E2 0, E3 0, E4 0}
LIN {X 572.549, Y 361.951, Z 400.98, A -110.612, B 84.801, C -94.37, E1 0, E2 0, E3 0, E4 0}
LIN {X 571.565, Y 362.231, Z 400.988, A -110.612, B 84.801, C -94.37, E1 0, E2 0, E3 0, E4 0}
LIN {X 571.396, Y 362.385, Z 400.98, A -110.612, B 84.801, C -94.37, E1 0, E2 0, E3 0, E4 0}
LIN {X 560.776, Y 364.467, Z 401.143, A -110.612, B 84.801, C -94.37, E1 0, E2 0, E3 0, E4 0}
LIN {X 559.908, Y 364.914, Z 401.133, A -110.612, B 84.801, C -94.37, E1 0, E2 0, E3 0, E4 0}
LIN {X 559.009, Y 364.986, Z 401.156, A -110.612, B 84.801, C -94.37, E1 0, E2 0, E3 0, E4 0}
LIN {X 558.479, Y 365.272, Z 401.148, A -110.612, B 84.801, C -94.37, E1 0, E2 0, E3 0, E4 0}
LIN {X 540.22, Y 368.452, Z 401.462, A -110.612, B 84.801, C -94.37, E1 0, E2 0, E3 0, E4 0}
LIN {X 540.126, Y 368.555, Z 401.456, A -110.612, B 84.801, C -94.37, E1 0, E2 0, E3 0, E4 0}
LIN {X 534.612, Y 369.495, Z 401.553, A -110.612, B 84.801, C -94.37, E1 0, E2 0, E3 0, E4 0}
LIN {X 533.295, Y 369.052, Z 401.633, A -110.612, B 84.801, C -94.37, E1 0, E2 0, E3 0, E4 0}
LIN {X 531.865, Y 369.73, Z 401.621, A -110.612, B 84.801, C -94.37, E1 0, E2 0, E3 0, E4 0}
LIN {X 529.601, Y 369.894, Z 401.679, A -110.612, B 84.801, C -94.37, E1 0, E2 0, E3 0, E4 0}
LIN {X 528.921, Y 369.452, Z 401.739, A -110.612, B 84.801, C -94.37, E1 0, E2 0, E3 0, E4 0}
LIN {X 526.892, Y 369.838, Z 401.771, A -110.612, B 84.801, C -94.37, E1 0, E2 0, E3 0, E4 0}
LIN {X 526.178, Y 370.535, Z 401.735, A -110.612, B 84.801, C -94.37, E1 0, E2 0, E3 0, E4 0}
LIN {X 524.831, Y 370.31, Z 401.797, A -110.612, B 84.801, C -94.37, E1 0, E2 0, E3 0, E4 0}
LIN {X 524.732, Y 370.324, Z 401.799, A -110.612, B 84.801, C -94.37, E1 0, E2 0, E3 0, E4 0}
LIN {X 523.139, Y 371.915, Z 401.714, A -110.612, B 84.801, C -94.37, E1 0, E2 0, E3 0, E4 0}
LIN {X 519.127, Y 372.655, Z 401.78, A -110.612, B 84.801, C -94.37, E1 0, E2 0, E3 0, E4 0}
LIN {X 517.966, Y 372.555, Z 401.825, A -110.612, B 84.801, C -94.37, E1 0, E2 0, E3 0, E4 0}
LIN {X 516.367, Y 372.864, Z 401.85, A -110.612, B 84.801, C -94.37, E1 0, E2 0, E3 0, E4 0}
LIN {X 515.551, Y 372.501, Z 401.907, A -110.612, B 84.801, C -94.37, E1 0, E2 0, E3 0, E4 0}
LIN {X 514.67, Y 371.453, Z 402.025, A -110.612, B 84.801, C -94.37, E1 0, E2 0, E3 0, E4 0}
LIN {X 505.664, Y 337.173, Z 405.233, A -110.612, B 84.801, C -94.37, E1 0, E2 0, E3 0, E4 0}
LIN {X 504.263, Y 330.85, Z 405.816, A -110.612, B 84.801, C -94.37, E1 0, E2 0, E3 0, E4 0}
LIN {X 593.753, Y 327.927, Z 403.199, A -110.612, B 84.801, C -94.37, E1 0, E2 0, E3 0, E4 0}
LIN {X 597.227, Y 343.546, Z 401.757, A -110.612, B 84.801, C -94.37, E1 0, E2 0, E3 0, E4 0}
LIN {X 587.328, Y 359.713, Z 400.697, A -110.612, B 84.801, C -94.37, E1 0, E2 0, E3 0, E4 0}
LIN {X 599.563, Y 356.145, Z 400.609, A -110.612, B 84.801, C -94.37, E1 0, E2 0, E3 0, E4 0}
LIN {X 599.29, Y 351.038, Z 401.053, A -110.612, B 84.801, C -94.37, E1 0, E2 0, E3 0, E4 0}
LIN {X 538.471, Y 368.776, Z 401.491, A -110.612, B 84.801, C -94.37, E1 0, E2 0, E3 0, E4 0}
LIN {X 514.261, Y 370.65, Z 402.106, A -110.612, B 84.801, C -94.37, E1 0, E2 0, E3 0, E4 0}
LIN {X 598.284, Y 346.144, Z 401.502, A -110.612, B 84.801, C -94.37, E1 0, E2 0, E3 0, E4 0}
LIN {X 597.105, Y 341.301, Z 401.952, A -110.612, B 84.801, C -94.37, E1 0, E2 0, E3 0, E4 0}
LIN {X 512.526, Y 365.969, Z 402.561, A -110.612, B 84.801, C -94.37, E1 0, E2 0, E3 0, E4 0}
LIN {X 510.836, Y 361.275, Z 403.015, A -110.612, B 84.801, C -94.37, E1 0, E2 0, E3 0, E4 0}
LIN {X 596.065, Y 336.417, Z 402.401, A -110.612, B 84.801, C -94.37, E1 0, E2 0, E3 0, E4 0}
LIN {X 595.071, Y 331.52, Z 402.85, A -110.612, B 84.801, C -94.37, E1 0, E2 0, E3 0, E4 0}
LIN {X 509.821, Y 356.384, Z 403.464, A -110.612, B 84.801, C -94.37, E1 0, E2 0, E3 0, E4 0}
LIN {X 508.846, Y 351.481, Z 403.912, A -110.612, B 84.801, C -94.37, E1 0, E2 0, E3 0, E4 0}
LIN {X 589.301, Y 328.016, Z 403.333, A -110.612, B 84.801, C -94.37, E1 0, E2 0, E3 0, E4 0}
LIN {X 567.227, Y 329.267, Z 403.934, A -110.612, B 84.801, C -94.37, E1 0, E2 0, E3 0, E4 0}
LIN {X 507.881, Y 346.576, Z 404.361, A -110.612, B 84.801, C -94.37, E1 0, E2 0, E3 0, E4 0}
LIN {X 506.891, Y 341.678, Z 404.81, A -110.612, B 84.801, C -94.37, E1 0, E2 0, E3 0, E4 0}
LIN {X 546.597, Y 330.097, Z 404.524, A -110.612, B 84.801, C -94.37, E1 0, E2 0, E3 0, E4 0}
LIN {X 528.454, Y 330.201, Z 405.096, A -110.612, B 84.801, C -94.37, E1 0, E2 0, E3 0, E4 0}
LIN {X 505.6, Y 336.867, Z 405.261, A -110.612, B 84.801, C -94.37, E1 0, E2 0, E3 0, E4 0}
LIN {X 504.543, Y 331.988, Z 405.71, A -110.612, B 84.801, C -94.37, E1 0, E2 0, E3 0, E4 0}
LIN {X 510.528, Y 330.243, Z 405.667, A -110.612, B 84.801, C -94.37, E1 0, E2 0, E3 0, E4 0}
LIN {X 597.208, Y 343.55, Z 401.758, A -110.612, B 84.801, C -94.37, E1 0, E2 0, E3 0, E4 0}
LIN {X 597.139, Y 343.365, Z 399.593, A -110.612, B 84.801, C -94.37, E1 0, E2 0, E3 0, E4 0}
LIN {X 594.204, Y 327.703, Z 401.02, A -110.612, B 84.801, C -94.37, E1 0, E2 0, E3 0, E4 0}
LIN {X 508.706, Y 330.19, Z 403.547, A -110.612, B 84.801, C -94.37, E1 0, E2 0, E3 0, E4 0}
LIN {X 504.72, Y 330.59, Z 403.641, A -110.612, B 84.801, C -94.37, E1 0, E2 0, E3 0, E4 0}
LIN {X 514.874, Y 369.912, Z 399.967, A -110.612, B 84.801, C -94.37, E1 0, E2 0, E3 0, E4 0}
LIN {X 515.676, Y 372.921, Z 399.685, A -110.612, B 84.801, C -94.37, E1 0, E2 0, E3 0, E4 0}
LIN {X 515.831, Y 372.979, Z 399.675, A -110.612, B 84.801, C -94.37, E1 0, E2 0, E3 0, E4 0}
LIN {X 518.025, Y 372.771, Z 399.622, A -110.612, B 84.801, C -94.37, E1 0, E2 0, E3 0, E4 0}
LIN {X 519.454, Y 371.759, Z 399.663, A -110.612, B 84.801, C -94.37, E1 0, E2 0, E3 0, E4 0}
LIN {X 521.59, Y 371.573, Z 399.61, A -110.612, B 84.801, C -94.37, E1 0, E2 0, E3 0, E4 0}
LIN {X 523.408, Y 370.904, Z 399.609, A -110.612, B 84.801, C -94.37, E1 0, E2 0, E3 0, E4 0}
LIN {X 523.901, Y 370.542, Z 399.624, A -110.612, B 84.801, C -94.37, E1 0, E2 0, E3 0, E4 0}
LIN {X 528.768, Y 369.677, Z 399.542, A -110.612, B 84.801, C -94.37, E1 0, E2 0, E3 0, E4 0}
LIN {X 528.853, Y 369.742, Z 399.533, A -110.612, B 84.801, C -94.37, E1 0, E2 0, E3 0, E4 0}
LIN {X 530.364, Y 370.047, Z 399.459, A -110.612, B 84.801, C -94.37, E1 0, E2 0, E3 0, E4 0}
LIN {X 530.49, Y 370.109, Z 399.45, A -110.612, B 84.801, C -94.37, E1 0, E2 0, E3 0, E4 0}
LIN {X 555.115, Y 365.541, Z 399.05, A -110.612, B 84.801, C -94.37, E1 0, E2 0, E3 0, E4 0}
LIN {X 556.091, Y 365.705, Z 399.005, A -110.612, B 84.801, C -94.37, E1 0, E2 0, E3 0, E4 0}
LIN {X 557.673, Y 365.31, Z 398.988, A -110.612, B 84.801, C -94.37, E1 0, E2 0, E3 0, E4 0}
LIN {X 559.307, Y 365.452, Z 398.923, A -110.612, B 84.801, C -94.37, E1 0, E2 0, E3 0, E4 0}
LIN {X 561.261, Y 364.645, Z 398.93, A -110.612, B 84.801, C -94.37, E1 0, E2 0, E3 0, E4 0}
LIN {X 569.484, Y 363.231, Z 398.787, A -110.612, B 84.801, C -94.37, E1 0, E2 0, E3 0, E4 0}
LIN {X 570.898, Y 362.238, Z 398.826, A -110.612, B 84.801, C -94.37, E1 0, E2 0, E3 0, E4 0}
LIN {X 570.926, Y 362.194, Z 398.829, A -110.612, B 84.801, C -94.37, E1 0, E2 0, E3 0, E4 0}
LIN {X 581.34, Y 360.25, Z 398.661, A -110.612, B 84.801, C -94.37, E1 0, E2 0, E3 0, E4 0}
LIN {X 582.796, Y 360.392, Z 398.602, A -110.612, B 84.801, C -94.37, E1 0, E2 0, E3 0, E4 0}
LIN {X 590.636, Y 358.924, Z 398.476, A -110.612, B 84.801, C -94.37, E1 0, E2 0, E3 0, E4 0}
LIN {X 591.268, Y 358.558, Z 398.487, A -110.612, B 84.801, C -94.37, E1 0, E2 0, E3 0, E4 0}
LIN {X 591.741, Y 358.52, Z 398.475, A -110.612, B 84.801, C -94.37, E1 0, E2 0, E3 0, E4 0}
LIN {X 592.002, Y 358.813, Z 398.442, A -110.612, B 84.801, C -94.37, E1 0, E2 0, E3 0, E4 0}
LIN {X 598.807, Y 357.19, Z 398.362, A -110.612, B 84.801, C -94.37, E1 0, E2 0, E3 0, E4 0}
LIN {X 598.921, Y 357.11, Z 398.365, A -110.612, B 84.801, C -94.37, E1 0, E2 0, E3 0, E4 0}
LIN {X 599.521, Y 356.079, Z 398.434, A -110.612, B 84.801, C -94.37, E1 0, E2 0, E3 0, E4 0}
LIN {X 597.139, Y 343.365, Z 399.593, A -110.612, B 84.801, C -94.37, E1 0, E2 0, E3 0, E4 0}
LIN {X 586.701, Y 359.692, Z 398.537, A -110.612, B 84.801, C -94.37, E1 0, E2 0, E3 0, E4 0}
LIN {X 599.52, Y 355.953, Z 398.444, A -110.612, B 84.801, C -94.37, E1 0, E2 0, E3 0, E4 0}
LIN {X 599.228, Y 350.851, Z 398.888, A -110.612, B 84.801, C -94.37, E1 0, E2 0, E3 0, E4 0}
LIN {X 535.28, Y 369.502, Z 399.348, A -110.612, B 84.801, C -94.37, E1 0, E2 0, E3 0, E4 0}
LIN {X 514.935, Y 370.249, Z 399.936, A -110.612, B 84.801, C -94.37, E1 0, E2 0, E3 0, E4 0}
LIN {X 598.27, Y 345.944, Z 399.337, A -110.612, B 84.801, C -94.37, E1 0, E2 0, E3 0, E4 0}
LIN {X 596.982, Y 341.132, Z 399.788, A -110.612, B 84.801, C -94.37, E1 0, E2 0, E3 0, E4 0}
LIN {X 512.784, Y 365.689, Z 400.393, A -110.612, B 84.801, C -94.37, E1 0, E2 0, E3 0, E4 0}
LIN {X 511.353, Y 360.919, Z 400.845, A -110.612, B 84.801, C -94.37, E1 0, E2 0, E3 0, E4 0}
LIN {X 596.095, Y 336.204, Z 400.236, A -110.612, B 84.801, C -94.37, E1 0, E2 0, E3 0, E4 0}
LIN {X 595.03, Y 331.327, Z 400.685, A -110.612, B 84.801, C -94.37, E1 0, E2 0, E3 0, E4 0}
LIN {X 510.172, Y 356.077, Z 401.296, A -110.612, B 84.801, C -94.37, E1 0, E2 0, E3 0, E4 0}
LIN {X 509.351, Y 351.129, Z 401.743, A -110.612, B 84.801, C -94.37, E1 0, E2 0, E3 0, E4 0}
LIN {X 589.212, Y 327.837, Z 401.169, A -110.612, B 84.801, C -94.37, E1 0, E2 0, E3 0, E4 0}
LIN {X 567.227, Y 329.062, Z 401.769, A -110.612, B 84.801, C -94.37, E1 0, E2 0, E3 0, E4 0}
